METHOD PRIVATE M_Errors : STRING(126)
VAR_INPUT
END_VAR
VAR_INST
END_VAR
CASE _AlarmNum OF	
1	: M_Errors :='1: INTERNAL error';	 	 
2	: M_Errors :='2: No Rtime';	 	 
3	: M_Errors :='3: Allocation locked memory error';	 	 
4	: M_Errors :='4: Insert mailbox error';
5	: M_Errors :='5: Wrong receive HMSG';	 	 
6	: M_Errors :='6: target port NOT found	ADS Server NOT started';	 
7	: M_Errors :='7: target machine NOT found Missing ADS routes';	 
8	: M_Errors :='8: Unknown command ID';	 	 
9	: M_Errors :='9: Bad task ID';	 	 
10	: M_Errors :='10: No IO';	 	 
11	: M_Errors :='11: Unknown ADS command';	 	 
12	: M_Errors :='12: Win 32 error';	 	 
13	: M_Errors :='13: Port NOT connected';	 	 
14	: M_Errors :='14: Invalid ADS length';	 	 
15	: M_Errors :='15: Invalid AMS Net ID';	 	 
16	: M_Errors :='16: Low Installation level';	 	 
17	: M_Errors :='17: No debug available';	 	 
18	: M_Errors :='18: Port disabled';	 	 
19	: M_Errors :='19: Port already connected';	 	 
20	: M_Errors :='20: ADS Sync Win32 error';	 	 
21	: M_Errors :='21: ADS Sync Timeout';	 	 
22	: M_Errors :='22: ADS Sync AMS error';	 	 
23	: M_Errors :='23: ADS Sync no index map';	 	 
24	: M_Errors :='24: Invalid ADS port';	 	 
25	: M_Errors :='25: No memory';	 	 
26	: M_Errors :='26: TCP send error';	 	 
27	: M_Errors :='27: Host unreachable	'; 	 
28	: M_Errors :='28: Invalid AMS fragment';
1101: M_Errors :='';
1792: M_Errors :='1792: error class <device error>';	 	 
1793: M_Errors :='1793: Service is NOT supported BY server';	 	 
1794: M_Errors :='1794: invalid index group';	 	 
1795: M_Errors :='1795: invalid index offset';	 	 
1796: M_Errors :='1796: reading/writing NOT permitted';	 	 
1797: M_Errors :='1797: parameter size NOT correct';	 	 
1798: M_Errors :='1798: invalid parameter value(S)';	 	 
1799: M_Errors :='1799: device is NOT in a ready state';	 	 
1800: M_Errors :='1800: device is busy';	 	 
1801: M_Errors :='1801: invalid context (must be in Windows)';	 	 
1802: M_Errors :='1802: out OF memory';	 	 
1803: M_Errors :='1803: invalid parameter value(S)';	 	 
1804: M_Errors :='1804: NOT found (files, ...)';	 	 
1805: M_Errors :='1805: syntax error in command OR file';	 	 
1806: M_Errors :='1806: objects DO NOT match';	 	 
1807: M_Errors :='1807: object already exists';	 	 
1808: M_Errors :='1808: symbol NOT found';	 	 
1809: M_Errors :='1809: symbol version invalid';	
1810: M_Errors :='1810: server is in invalid state';	 	 
1811: M_Errors :='1811: AdsTransMode NOT supported';	 	 
1812: M_Errors :='1812: notification handle is invalid';	
1813: M_Errors :='1813: notification client NOT registered';	 	 
1814: M_Errors :='1814: no more notification handles';	 	 
1815: M_Errors :='1815: size FOR watch too big';	 	 
1816: M_Errors :='1816: device NOT initialized';	 	 
1817: M_Errors :='1817: device has a timeout';	 	 
1818: M_Errors :='1818: query INTERFACE failed';	 	 
1819: M_Errors :='1819: wrong INTERFACE required';	 	 
1820: M_Errors :='1820: class ID is invalid';	 	 
1821: M_Errors :='1821: object ID is invalid';	 	 
1822: M_Errors :='1822: request is pending';	 	 
1823: M_Errors :='1823: request is aborted';	 	 
1824: M_Errors :='1824: signal warning';	 	 
1825: M_Errors :='1825: invalid ARRAY index';	 	 
1826: M_Errors :='1826: symbol NOT active';	
1827: M_Errors :='1827: access denied';	 	 
1828: M_Errors :='1828: missing license';	 	
1836: M_Errors :='1836: exception occured during system start';	
1856: M_Errors :='1856: Error class <client error>';	 	 
1857: M_Errors :='1857: invalid parameter AT service';	 	 
1858: M_Errors :='1858: polling list is empty';	 	 
1859: M_Errors :='1859: VAR connection already in use';	 	 
1860: M_Errors :='1860: invoke ID in use';	 	 
1861: M_Errors :='1861: timeout elapsed'; 	
1862: M_Errors :='1862: error in win32 subsystem';	 	 
1863: M_Errors :='1863: Invalid client timeout value';	 	 
1864: M_Errors :='1864: ads-port NOT opened';	 	 
1872: M_Errors :='1872: INTERNAL error in ads sync';	 	 
1873: M_Errors :='1873: hash table overflow';	 	 
1874: M_Errors :='1874: key NOT found in hash';	 	 
1875: M_Errors :='1875: no more symbols in cache';	 	 
1876: M_Errors :='1876: invalid response received';	 	 
1877: M_Errors :='1877: sync port is locked';
4096:  M_Errors:=' 4096: INTERNAL error in the REAL-TIME system.';
4097:  M_Errors:=' 4097: Timer value is NOT valid.';
4098:  M_Errors:=' 4098: Task POINTER has the invalid value 0 (zero).';
4099:  M_Errors:=' 4099: Stack POINTER has the invalid value 0 (zero).';
4100:  M_Errors:=' 4100: The request task priority is already assigned.';
4101:  M_Errors:=' 4101: No free TCB (Task Control Block) available. The maximum number OF TCBs is 64.';
4102:  M_Errors:=' 4102: No free semaphores available. The maximum number OF semaphores is 64.';
4103:  M_Errors:=' 4103: No free space available in the queue. The maximum number OF positions in the queue is 64.';
4109:  M_Errors:=' 4109: An external synchronization interrupt is already applied.';
4110:  M_Errors:=' 4110: No external sync interrupt applied.';
4111:  M_Errors:=' 4111: Application OF the external synchronization interrupt has failed.';
4112:  M_Errors:=' 4112: Call OF a service FUNCTION in the wrong context';
4119:  M_Errors:=' 4119: Intel VT-x extension is NOT supported.';
4120:  M_Errors:=' 4120: Intel VT-x extension is NOT enabled in the BIOS.';
4121:  M_Errors:=' 4121: Missing FUNCTION in Intel VT-x extension.';
4122:  M_Errors:=' 4122: Activation OF Intel VT-x fails.';
16384: M_Errors :='16384: INTERNAL error';
16385: M_Errors :='16385: Memory error';
16386: M_Errors :='16386: Nc RETAIN data error (PERSISTENT data)';
16387: M_Errors :='16387: Parameter FOR Monitoring the NC Setpoint Issuing is Invalid';
16388: M_Errors :='16388: External Error';
16400: M_Errors :='16400: Channel identifier NOT allowed';
16401: M_Errors :='16401: Group identifier NOT allowed';
16402: M_Errors :='16402: Axis identifier NOT allowed';
16403: M_Errors :='16403: Encoder identifier NOT allowed';
16404: M_Errors :='16404: Controller identifier NOT allowed';
16405: M_Errors :='16405: Drive identifier NOT allowed';
16406: M_Errors :='16406: Table identifier NOT allowed';
16416: M_Errors :='16416: No PLC-axis INTERFACE during creation OF an axis';
16417: M_Errors :='16417: No axis-PLC INTERFACE during creation OF an axis';
16418: M_Errors :='16418: No encoder-I/O INTERFACE during creation OF an axis';
16419: M_Errors :='16419: No I/O-encoder INTERFACE during creation OF an axis';
16420: M_Errors :='16420: INTERNAL No drive-I/O INTERFACE during creation OF an axis';
16421: M_Errors :='16421: INTERNAL No I/O-drive INTERFACE during creation OF an axis';
16432: M_Errors :='16432: Coupling TYPE NOT allowed';
16434: M_Errors :='16434: Parameter Unknown Channel TYPE';
16448: M_Errors :='16448: Axis is incompatible';
16464: M_Errors :='16464: Channel NOT ready FOR operation';
16465: M_Errors :='16465: Group NOT ready FOR operation';
16466: M_Errors :='16466: Axis NOT ready FOR operation';
16480: M_Errors :='16480: Channel exists';
16481: M_Errors :='16481: Group exists';
16482: M_Errors :='16482: Axis exists';
16483: M_Errors :='16483: Table exists';
16496: M_Errors :='16496: Axis index NOT allowed';
16497: M_Errors :='16497: Axis index NOT allowed';
16641: M_Errors :='16641: Group index NOT allowed';
16642: M_Errors :='16642: Null POINTER';
16643: M_Errors :='16643: No process image';
16644: M_Errors :='16644: M-FUNCTION index NOT allowed';
16645: M_Errors :='16645: No memory';
16646: M_Errors :='16646: NOT ready';
16647: M_Errors :='16647: FUNCTION/command NOT supported';
16648: M_Errors :='16648: Invalid parameter WHILE starting';
16649: M_Errors :='16649: Channel FUNCTION/command NOT executable';
16650: M_Errors :='16650: ItpGoAhead NOT executable';
16656: M_Errors :='16656: Error opening a file';
16657: M_Errors :='16657: Syntax error during loading';
16658: M_Errors :='16658: Syntax error during interpretation';
16659: M_Errors :='16659: Missing subroutine';
16660: M_Errors :='16660: Loading buffer OF interpreter is too small';
16661: M_Errors :='16661: Symbolic - reserved';
16662: M_Errors :='16662: Symbolic - reserved';
16663: M_Errors :='16663: Subroutine incomplete';
16664: M_Errors :='16664: Error WHILE loading the NC PROGRAM';
16665: M_Errors :='16665: Error WHILE loading the NC PROGRAM';
16672: M_Errors :='16672: Divide BY zero';
16673: M_Errors :='16673: Invalid circle parameterization';
16674: M_Errors :='16674: Invalid FPU-Operation';
16688: M_Errors :='16688: Stack overflow: subroutines';
16689: M_Errors :='16689: Stack underflow: subroutines';
16690: M_Errors :='16690: Stack overflow: arithmetic unit';
16691: M_Errors :='16691: Stack underflow: arithmetic unit';
16704: M_Errors :='16704: Register index NOT allowed';
16705: M_Errors :='16705: Unacceptable G-FUNCTION index';
16706: M_Errors :='16706: Unacceptable M-FUNCTION index';
16707: M_Errors :='16707: Unacceptable extended address';
16708: M_Errors :='16708: Unacceptable index TO the INTERNAL H-FUNCTION';
16709: M_Errors :='16709: Machine data value unacceptable';
16720: M_Errors :='16720: Cannot change tool PARAMS here';
16721: M_Errors :='16721: Cannot calculate tool compensation';
16722: M_Errors :='16722: The plane FOR the tool compensation cannot be changed here';
16723: M_Errors :='16723: The D-WORD is missing OR invalid BY turning on the tool compensation';
16724: M_Errors :='16724: The specified tool radius is invalid because the value is <= zero';
16725: M_Errors :='16725: The tool radius cannot be changed here';
16726: M_Errors :='16726: Collision Detection Table is full';
16727: M_Errors :='16727: INTERNAL error WHILE turning on the contour collision detection';
16728: M_Errors :='16728: INTERNAL error within the contour collision detection: update reversed geo failed';
16729: M_Errors :='16729: Unexpected combination OF geometry types BY active contour collision detection';
16730: M_Errors :='16730: Programmed inner circle is smaller than the cutter radius';
16731: M_Errors :='16731: Bottle neck detection recognized contour violation';
16732: M_Errors :='16732: Table FOR corrected entries is full';
16733: M_Errors :='16733: Input table FOR tangential following is full';
16734: M_Errors :='16734: Executing table FOR tangential following is full';
16735: M_Errors :='16735: Geometric entry FOR tangential following cannot be calculated';
16736: M_Errors :='16736: INTERNAL reserved';
16737: M_Errors :='16737: INTERNAL reserved';
16738: M_Errors :='16738: The actual active interpolation rules, zeroshifts, OR rotation cannot be detected';
16752: M_Errors :='16752: Error WHILE loading: Invalid parameter';
16753: M_Errors :='16753: Invalid contour start position';
16754: M_Errors :='16754: Retrace: Invalid INTERNAL entry index';
16755: M_Errors :='16755: Invalid G Code';
16756: M_Errors :='16756: Error WHILE Opening the G Code File';
16896: M_Errors :='16896: Group ID NOT allowed';
16897: M_Errors :='16897: Group TYPE NOT allowed';
16898: M_Errors :='16898: Master axis index NOT allowed';
16899: M_Errors :='16899: Slave axis index NOT ';
16900: M_Errors :='16900: Initializing INTERNAL Error';
16901: M_Errors :='16901: Invalid cycle TIME FOR statement execution task (SAF)';
16903: M_Errors :='16903: Invalid cycle TIME FOR the statement preparation task(SVB)';
16904: M_Errors :='16904: Single step mode NOT allowed';
16905: M_Errors :='16905: Group deactivation NOT allowed';
16906: M_Errors :='16906: Initialization Statement execution state (SAF state) NOT allowed';
16907: M_Errors :='16907: Channel address';
16908: M_Errors :='16908: Axis address (master axis)';
16909: M_Errors :='16909: Master axis address';
16910: M_Errors :='16910: Slave axis address';
16911: M_Errors :='16911: Slave set value generator address';
16912: M_Errors :='16912: Encoder address';
16913: M_Errors :='16913: Controller address';
16914: M_Errors :='16914: Drive address';
16915: M_Errors :='16915: Address Address Master Setpoint Generator';
16916: M_Errors :='16916: Axis INTERFACE NC TO PLC address';
16917: M_Errors :='16917: Slave axis address';
16918: M_Errors :='16918: Table address unknown';
16919: M_Errors :='16919: NcControl address';
16920: M_Errors :='16920: Axis is blocked FOR commands WHILE PERSISTENT NC data are queued';
16921: M_Errors :='16921: The scaling mode MASTER-AUTO-OFFSET is invalid because no REFERENCE table was found';
16922: M_Errors :='16922: The master axis start position does NOT permit synchronization';
16923: M_Errors :='16923: Slave coupling factor (gearing factor) OF 0.0 is NOT allowed';
16924: M_Errors :='16924: Insertion OF master axis into group NOT allowed';
16925: M_Errors :='16925: Deletion OF master axis FROM group NOT allowed'; 
16926: M_Errors :='16926: FUNCTION/feature is NOT supported FROM the setpoint generator';
16927: M_Errors :='16927: Group initialization';
16928: M_Errors :='16928: Group NOT ready / group NOT ready FOR new task';
16929: M_Errors :='16929: Requested set velocity is NOT allowed';
16930: M_Errors :='16930: Requested target position is NOT allowed (master axis)';
16931: M_Errors :='16931: No enable FOR controller AND/OR feed (Master axis)';
16932: M_Errors :='16932: Movement smaller than one encoder increment';
16933: M_Errors :='16933: Drive NOT ready during axis start';
16934: M_Errors :='16934: Invalid parameters OF the emergency stop.';
16935: M_Errors :='16935: The setpoint generator is inactive such that no instructions are accepted';
16936: M_Errors :='16936: Requested traverse distance is NOT allowed';
16937: M_Errors :='16937: Requested target position is NOT allowed (slave axis)';
16938: M_Errors :='16938: No enable FOR controller AND/OR feed (slave axis)';
16939: M_Errors :='16939: The activation position (position threshold) is out OF range OF the actual positioning';
16940: M_Errors :='16940: The start OR activation data OF the external setpoint generation are NOT valid';
16941: M_Errors :='16941: Velocity is NOT CONSTANT';
16942: M_Errors :='16942: Jerk less than OR equal TO 0.0 is NOT allowed';
16943: M_Errors :='16943: Acceleration less than OR equal TO 0.0 is NOT allowed';
16944: M_Errors :='16944: Absolute deceleration value less than OR equal TO 0.0 is NOT allowed';
16945: M_Errors :='16945: Set velocity less than OR equal TO 0.0 is NOT allowed';
16946: M_Errors :='16946: Loss OF precision when trying a positioning';
16947: M_Errors :='16947: Cycle TIME less than OR equal TO 0.0 is NOT allowed';
16948: M_Errors :='16948: PTP data TYPE <intasdouble> range exceeded';
16949: M_Errors :='16949: PTP LHL velocity profile cannot be generated';
16950: M_Errors :='16950: PTP HML velocity profile cannot be generated';
16951: M_Errors :='16951: Start data address is invalid';
16952: M_Errors :='16952: Velocity override (start override) is NOT allowed';
16953: M_Errors :='16953: Start TYPE NOT allowed';
16954: M_Errors :='16954: Velocity overflow (overshoot in the velocity)';
16955: M_Errors :='16955: Start parameter FOR the axis structure is invalid';
16956: M_Errors :='16956: Override generator initialization parameter invalid';
16957: M_Errors :='16957: Slave axis has NOT set value generator';
16958: M_Errors :='16958: Table is empty';
16959: M_Errors :='16959: Table is full';
16960: M_Errors :='16960: No memory available';
16961: M_Errors :='16961: Table already contains an entry';
16962: M_Errors :='16962: Stop is already active';
16963: M_Errors :='16963: Compensation has NOT been carried out over the full compensation section';
16964: M_Errors :='16964: INTERNAL parameters FOR the compensation are invalid';
16965: M_Errors :='16965: Compensation active';
16966: M_Errors :='16966: Compensation NOT active';
16967: M_Errors :='16967: Compensation TYPE invalid';
16968: M_Errors :='16968: Axis address FOR compensation invalid';
16969: M_Errors :='16969: Invalid slave address';
16970: M_Errors :='16970: Coupling velocity invalid';
16971: M_Errors :='16971: Coupling velocities NOT CONSTANT';
16972: M_Errors :='16972: Cycle TIME less than OR equal TO 0.0 is NOT allowed';
16973: M_Errors :='16973: Decoupling task NOT allowed';
16974: M_Errors :='16974: FUNCTION NOT allowed';
16975: M_Errors :='16975: No valid table weighting has been set';
16976: M_Errors :='16976: Axis TYPE, actual position TYPE OR end position TYPE is NOT allowed';
16977: M_Errors :='16977: FUNCTION NOT presently supported';
16978: M_Errors :='16978: State OF state machine invalid';
16979: M_Errors :='16979: REFERENCE cam became free too soon';
16980: M_Errors :='16980: Clearance monitoring between activation OF the hardware latch AND appearance OF the sync pulse';
16981: M_Errors :='16981: No memory available';
16982: M_Errors :='16982: The table slave axis has no active table';
16983: M_Errors :='16983: FUNCTION NOT allowed';
16984: M_Errors :='16984: Stopping compensation NOT allowed';
16985: M_Errors :='16985: Slave table is being used';
16986: M_Errors :='16986: Master OR slave axis is processing a job WHILE coupling is requested';
16987: M_Errors :='16987: Slave (start) parameter is incorrect';
16988: M_Errors :='16988: Slave TYPE is incorrect';
16989: M_Errors :='16989: Axis stop is already active';
16990: M_Errors :='16990: Maximum number OF tables per slave generator reached';
16991: M_Errors :='16991: The scaling mode is invalid';
16992: M_Errors :='16992: Controller enable NOT present';
16993: M_Errors :='16993: Table NOT found';
16994: M_Errors :='16994: Incorrect table TYPE';
16995: M_Errors :='16995: Single step mode';
16996: M_Errors :='16996: Group task unknown (asynchronous table entry)';
16997: M_Errors :='16997: Group FUNCTION unknown (synchronous FUNCTION)';
16998: M_Errors :='16998: Group task FOR slave NOT allowed';
16999: M_Errors :='16999: Group FUNCTION FOR slave NOT allowed';
17000: M_Errors :='17000: FUNCTION NCI Setpoint Generator is Inactive';
17001: M_Errors :='17001: Startposition=Setpoint Position';
17002: M_Errors :='17002: Parameters OF the delay-generator are invalid';
17003: M_Errors :='17003: External parameters OF the superimposed instruction are invalid';
17004: M_Errors :='17004: Invalid override TYPE.';
17005: M_Errors :='17005: Activation position under/overrun';
17006: M_Errors :='17006: Activation impossible: Master is standing';
17007: M_Errors :='17007: Activation mode NOT possible';
17008: M_Errors :='17008: Start parameter FOR the compensation is invalid';
17009: M_Errors :='17009: Start parameter FOR the compensation is invalid';
17010: M_Errors :='17010: Start parameter FOR the compensation is invalid';
17011: M_Errors :='17011: Target position under/overrun';
17012: M_Errors :='17012: Target position will be under/overrun';
17013: M_Errors :='17013: Parameter Group Parameter is Invalid';
17014: M_Errors :='17014: Monitoring Joint Error AT Start OF Setpoint Generation';
17015: M_Errors :='17015: Dynamic parameters NOT permitted';
17017: M_Errors :='17017: The New Target';
17018: M_Errors :='17018: New Velocity FOR Moving OR the FINAL Target Velocity is Invalid';
17019: M_Errors :='17019: The FINAL Velocity OR the New Target Position is Invalid';
17020: M_Errors :='17020: The New Moving Velocity is Invalid';
17021: M_Errors :='17021: INTERNAL Starting Mode is Invalid';
17022: M_Errors :='17022: A requested motion command could NOT be realized';
17023: M_Errors :='17023: The new target position either has been overrun OR will be overrun';
17024: M_Errors :='17024: Group NOT ready / group NOT ready FOR new task';
17025: M_Errors :='17025: The parameters OF the oriented stop (O-Stop) are NOT admitted.';
17026: M_Errors :='17026: The modulo target position OF the modulo-start is invalid';
17027: M_Errors :='17027: The online change activation mode is invalid';
17028: M_Errors :='17028: The parameterized jerk rate is NOT permitted';
17029: M_Errors :='17029: The parameterized acceleration OR deceleration is NOT permitted';
17030: M_Errors :='17030: The parameterized velocity is NOT permitted';
17031: M_Errors :='17031: A activation cannot be executed due TO a pending activation';
17032: M_Errors :='17032: Illegal combination OF different cycle times within an axis group';
17033: M_Errors :='17033: Illegal motion reversal';
17034: M_Errors :='17034: Illegal moment FOR an axis command because there is an old axis command active';
17035: M_Errors :='17035: Error in the stop-calculation routine';
17036: M_Errors :='17036: A command with activation position cannot be performed because the remaining path is too short';
17037: M_Errors :='17037: Illegal decouple TYPE when decoupling a slave axis';
17038: M_Errors :='17038: Illegal target velocity when decoupling a slave axis';
17039: M_Errors :='17039: The command new dynamic parameter cannot be performed since THIS would require a new target velocity';
17040: M_Errors :='17040: A command with activation position cannot be performed because the axis is already in the brake phase';
17041: M_Errors :='17041: Decouple routine OF slave axis does NOT RETURN a valid solution';
17042: M_Errors :='17042: Command NOT be executed because the command buffer is full filled';
17043: M_Errors :='17043: Command is rejected due TO an INTERNAL error in the Look Ahead';
17044: M_Errors :='17044: Command is rejected because the segment target velocity is NOT realized';
17045: M_Errors :='17045: Successive commands have the same FINAL position';
17046: M_Errors :='17046: Logical positioning direction is inconsistent with the direction OF the buffer command';
17047: M_Errors :='17047: Command is rejected because the remaining positioning length is TO small';
17050: M_Errors :='17050: FUNCTION Restart has Failed';
17051: M_Errors :='17051: Collect error FOR invalid start parameters';
17052: M_Errors :='17052: REFERENCE cam is NOT found';
17053: M_Errors :='17053: REFERENCE cam became NOT free';
17054: M_Errors :='17054: IO sync pulse was NOT found (only when using hardware latch)';
17055: M_Errors :='17055: The Used Buffer Mode is Unknown OR NOT Supported in THIS Context';
17056: M_Errors :='17056: Group/axis consequential error';
17057: M_Errors :='17057: Velocity reduction factor FOR C0/C1 transition is NOT allowed';
17058: M_Errors :='17058: Critical angle AT segment transition NOT allowed';
17059: M_Errors :='17059: Radius OF the tolerance sphere';
17060: M_Errors :='17060: Parameter NOT implemented';
17061: M_Errors :='17061: Start TYPE';
17062: M_Errors :='17062: Parameter NOT implemented';
17063: M_Errors :='17063: Blending with given parameters NOT possible';
17064: M_Errors :='17064: Parameter NOT implemented';
17065: M_Errors :='17065: Curve velocity reduction METHOD NOT allowed';
17066: M_Errors :='17066: Minimum velocity NOT allowed';
17067: M_Errors :='17067: Power FUNCTION input NOT allowed';
17068: M_Errors :='17068: Dynamic change parameter NOT allowed';
17069: M_Errors :='17069: Memory allocation error';
17070: M_Errors :='17070: The calculated end position differs FROM the end position in the nc instruction';
17071: M_Errors :='17071: Calculate remaining chord length';
17072: M_Errors :='17072: Set value generator SVB active';
17073: M_Errors :='17073: SVB parameter NOT allowed';
17074: M_Errors :='17074: Velocity reduction factor NOT allowed';
17075: M_Errors :='17075: Helix is a circle';
17076: M_Errors :='17076: Helix is a straight line';
17077: M_Errors :='17077: Guider parameter NOT allowed';
17078: M_Errors :='17078: Invalid segment address';
17079: M_Errors :='17079: Unparameterized generator';
17080: M_Errors :='17080: Unparameterized table';
17082: M_Errors :='17082: The calculation OF the arc length OF the smoothed path failed (INTERNAL error)';
17083: M_Errors :='17083: The radius OF the tolerance ball is too small (smaller than 0.1 mm)';
17084: M_Errors :='17084: INTERNAL Error WHILE calculating DXD-Software-LIMIT switches (INTERNAL error)';
17085: M_Errors :='17085: NC-Block violates software LIMIT switches OF the group';
17086: M_Errors :='17086: INTERNAL error in the evaluation OF a possible software LIMIT switch violation';
17087: M_Errors :='17087: Invalid REFERENCE speed TYPE';
17088: M_Errors :='17088: Interpolating group contains axes OF an incorrect axis TYPE';
17089: M_Errors :='17089: Scalar product cannot be calculated';
17090: M_Errors :='17090: Inverse cosine cannot be calculated';
17091: M_Errors :='17091: Invalid table entry TYPE';
17092: M_Errors :='17092: Invalid DIN66025 information TYPE';
17093: M_Errors :='17093: Invalid dimension';
17094: M_Errors :='17094: Geometrical object is NOT a straight line';
17095: M_Errors :='17095: Geometrical object is NOT a circle';
17096: M_Errors :='17096: Geometrical object is NOT a helix';
17097: M_Errors :='17097: Set velocity less than OR equal TO 0.0 is invalid';
17098: M_Errors :='17098: Address FOR look-ahead invalid';
17099: M_Errors :='17099: Set value generator SAF active';
17100: M_Errors :='17100: CNC set value generation NOT active';
17101: M_Errors :='17101: CNC set value generation in the stop phase';
17102: M_Errors :='17102: Override NOT allowed';
17103: M_Errors :='17103: Invalid table address';
17104: M_Errors :='17104: Invalid table entry TYPE';
17105: M_Errors :='17105: Memory allocation failed';
17106: M_Errors :='17106: Memory allocation failed';
17107: M_Errors :='17107: Invalid parameter';
17108: M_Errors :='17108: Delete Distance TO Go failed';
17109: M_Errors :='17109: The setpoint generator OF the flying saw generates incompatible values (INTERNAL error)';
17110: M_Errors :='17110: Axis will be stopped since otherwise it will overrun its target position';
17111: M_Errors :='17111: INTERNAL error in the transformation FROM slave TO master';
17112: M_Errors :='17112: Wrong direction in the transformation OF slave TO master';
17114: M_Errors :='17114: Parameter OF Motion FUNCTION (MF) table incorrect';
17115: M_Errors :='17115: Parameter OF Motion FUNCTION (MF) table incorrect';
17116: M_Errors :='17116: INTERNAL error BY using Motion FUNCTION (MF)';
17117: M_Errors :='17117: Axis coupling with synchronization generator declined because OF incorrect axis dynamic values';
17118: M_Errors :='17118: Coupling conditions OF synchronization generator incorrect';
17119: M_Errors :='17119: Moving profile OF synchronization generator declines dynamic LIMIT OF slave axis';
17120: M_Errors :='17120: Invalid parameter';
17121: M_Errors :='17121: Invalid parameter';
17122: M_Errors :='17122: External generator is active';
17123: M_Errors :='17123: External generator is NOT active';
17124: M_Errors :='17124: NC-Block with auxiliary axis violates software LIMIT switches OF the group';
17125: M_Errors :='17125: NC-Block TYPE Bezier spline curve contains a cusp (singularity)';
17127: M_Errors :='17127: Value FOR dead TIME compensation NOT allowed';
17128: M_Errors :='17128: GROUPERR_RANGE_NOMOTIONWINDOW';
17129: M_Errors :='17129: GROUPERR_RANGE_NOMOTIONFILTERTIME';
17130: M_Errors :='17130: GROUPERR_RANGE_TIMEUNITFIFO';
17131: M_Errors :='17131: GROUPERR_RANGE_OVERRIDETYPE';
17132: M_Errors :='17132: GROUPERR_RANGE_OVERRIDECHANGETIME';
17133: M_Errors :='17133: GROUPERR_FIFO_INVALIDDIMENSION';
17134: M_Errors :='17134: GROUPERR_ADDR_FIFOTABLE';
17135: M_Errors :='17135: Axis is locked FOR motion commands because a stop command is still active';
17136: M_Errors :='17136: Invalid number OF auxiliary axes';
17137: M_Errors :='17137: Invalid reduction parameter FOR auxiliary axes';
17138: M_Errors :='17138: Invalid dynamic parameter FOR auxiliary axes';
17139: M_Errors :='17139: Invalid coupling parameter FOR auxiliary axes';
17140: M_Errors :='17140: Invalid auxiliary axis entry';
17142: M_Errors :='17142: Invalid parameter';
17144: M_Errors :='17144: Block search - segment NOT found';
17145: M_Errors :='17145: Blocksearch - invalid remaining segment length';
17147: M_Errors :='17147: INTERNAL INTERNAL Error in the Context OF Coupled Axes (Slave Axes)';
17148: M_Errors :='17148: Parameter Parameter FOR the Maximum Number OF Jobs (Entries) TO be Transferred is Invalid';
17151: M_Errors :='17151: Monitoring Customer Specific Error';
17152: M_Errors :='17152: Axis ID NOT allowed';
17153: M_Errors :='17153: Axis TYPE NOT allowed';
17158: M_Errors :='17158: Slow manual velocity NOT allowed';
17159: M_Errors :='17159: Fast manual velocity NOT allowed';
17160: M_Errors :='17160: High speed NOT allowed';
17161: M_Errors :='17161: Acceleration NOT allowed';
17162: M_Errors :='17162: Deceleration NOT allowed';
17163: M_Errors :='17163: Jerk NOT allowed';
17164: M_Errors :='17164: Delay TIME between position AND velocity is NOT allowed';
17165: M_Errors :='17165: Override-TYPE NOT allowed';
17166: M_Errors :='17166: NCI: Velo-Jump-Factor NOT allowed';
17167: M_Errors :='17167: NCI: Radius OF tolerance sphere FOR the auxiliary axes is invalid';
17168: M_Errors :='17168: NCI: Value FOR maximum deviation FOR the auxiliary axes is invalid';
17170: M_Errors :='17170: Referencing velocity in direction OF cam NOT allowed';
17171: M_Errors :='17171: Referencing velocity in sync direction NOT allowed';
17172: M_Errors :='17172: Pulse width in positive direction NOT allowed';
17173: M_Errors :='17173: Pulse width in negative direction NOT allowed';
17174: M_Errors :='17174: Pulse TIME in positive direction NOT allowed';
17175: M_Errors :='17175: Pulse TIME in negative direction NOT allowed';
17176: M_Errors :='17176: Creep distance in positive direction NOT allowed';
17177: M_Errors :='17177: Creep distance in negative direction NOT allowed';
17178: M_Errors :='17178: Braking distance in positive direction NOT allowed';
17179: M_Errors :='17179: Braking distance in negative direction NOT allowed';
17180: M_Errors :='17180: Braking TIME in positive direction NOT allowed';
17181: M_Errors :='17181: Braking TIME in negative direction NOT allowed';
17182: M_Errors :='17182: Switching TIME FROM high TO low speed NOT allowed';
17183: M_Errors :='17183: Creep distance FOR stop NOT allowed';
17184: M_Errors :='17184: Motion monitoring NOT allowed';
17185: M_Errors :='17185: Position window monitoring NOT allowed';
17186: M_Errors :='17186: Target window monitoring NOT allowed';
17187: M_Errors :='17187: Loop NOT allowed';
17188: M_Errors :='17188: Motion monitoring TIME NOT allowed';
17189: M_Errors :='17189: Target window range NOT allowed';
17190: M_Errors :='17190: Position window range NOT allowed';
17191: M_Errors :='17191: Position window monitoring TIME NOT allowed';
17192: M_Errors :='17192: Loop movement NOT allowed';
17193: M_Errors :='17193: Axis cycle TIME NOT allowed';
17194: M_Errors :='17194: Stepper motor operating mode NOT allowed';
17195: M_Errors :='17195: Displacement per stepper motor step NOT allowed';
17196: M_Errors :='17196: Minimum speed FOR stepper motor set value profile NOT allowed';
17197: M_Errors :='17197: Stepper motor stages FOR one speed stage NOT allowed';
17198: M_Errors :='17198: DWORD FOR the interpretation OF the axis units NOT allowed';
17199: M_Errors :='17199: Maximum velocity NOT allowed';
17200: M_Errors :='17200: Motion monitoring window NOT allowed';
17201: M_Errors :='17201: PEH TIME monitoring NOT allowed';
17202: M_Errors :='17202: PEH monitoring TIME NOT allowed';
17203: M_Errors :='17203: Parameter Break Release Delay is Invalid';
17204: M_Errors :='17204: Parameter NC Data Persistence is Invalid';
17205: M_Errors :='17205: Parameter FOR the Error Reaction Mode is Invalid';
17206: M_Errors :='17206: Parameter FOR the Error Reaction Delay is Invalid';
17207: M_Errors :='17207: Parameter “Couple Slave TO Actual Values IF NOT Enabled” is Invalid';
17208: M_Errors :='17208: Parameter Allow Motion Commands TO Slave Axis” is Invalid';
17209: M_Errors :='17209: Parameter Parameter “Allow Motion Commands TO External Setpoint Axis” is Invalid';
17210: M_Errors :='17210: Parameter Parameter “Fading Acceleration” is Invalid';
17211: M_Errors :='17211: Fast Axis Stop Signal TYPE NOT allowed';
17216: M_Errors :='17216: Initialization Parameter Axis initialization';
17217: M_Errors :='17217: Address Parameter Group address';
17218: M_Errors :='17218: Address Parameter Encoder address';
17219: M_Errors :='17219: Address Parameter Controller address';
17220: M_Errors :='17220: Address Parameter Drive address';
17221: M_Errors :='17221: Address Parameter Axis INTERFACE PLC TO NC address';
17222: M_Errors :='17222: Address Parameter Axis INTERFACE NC TO PLC address';
17223: M_Errors :='17223: Address Parameter Size OF axis INTERFACE NC TO PLC is NOT allowed';
17224: M_Errors :='17224: Address Parameter Size OF axis INTERFACE PLC TO NC is NOT allowed';
17238: M_Errors :='17238: Monitoring Parameter Controller enable';
17239: M_Errors :='17239: There is no feed enable FOR negative motion direction';
17240: M_Errors :='17240: Monitoring Parameter Feed enable plus';
17241: M_Errors :='17241: Monitoring Parameter Set velocity NOT allowed';
17242: M_Errors :='17242: Monitoring Parameter Movement smaller than one encoder increment';
17243: M_Errors :='17243: Monitoring Parameter Set acceleration monitoring';
17244: M_Errors :='17244: Monitoring Parameter PEH TIME monitoring';
17245: M_Errors :='17245: Monitoring Parameter Encoder existence monitoring / movement monitoring';
17246: M_Errors :='17246: Monitoring Parameter Looping distance less than breaking distance';
17247: M_Errors :='17247: Monitoring Starting Velocity Invalid';
17248: M_Errors :='17248: Monitoring FINAL Velocity Invalid';
17249: M_Errors :='17249: Monitoring Parameter TIME range exceeded (future)';
17250: M_Errors :='17250: Monitoring Parameter TIME range exceeded (past)';
17251: M_Errors :='17251: Monitoring Parameter Position cannot be determined';
17252: M_Errors :='17252: Monitoring Parameter Position indeterminable (conflicting direction OF travel)';
17264: M_Errors :='17264: Monitoring No Slave Coupling Possible (Velocity Violation)';
17265: M_Errors :='17265: Monitoring No Slave Coupling Possible (Acceleration Violation)';
17266: M_Errors :='17266: Monitoring FINAL Velocity invalid';
17312: M_Errors :='17312: INTERNAL Parameter Axis consequential error';
17408: M_Errors :='17408: Encoder ID NOT allowed';
17409: M_Errors :='17409: Encoder TYPE NOT allowed';
17410: M_Errors :='17410: Encoder mode';
17411: M_Errors :='17411: Encoder counting direction inverted?';
17412: M_Errors :='17412: Referencing status';
17413: M_Errors :='17413: Encoder increments FOR each physical encoder rotation';
17414: M_Errors :='17414: Scaling factor';
17415: M_Errors :='17415: Position offset (zero point offset)';
17416: M_Errors :='17416: Modulo factor';
17417: M_Errors :='17417: Position filter TIME';
17418: M_Errors :='17418: Velocity filter TIME';
17419: M_Errors :='17419: Acceleration filter TIME';
17420: M_Errors :='17420: Cycle TIME NOT allowed';
17422: M_Errors :='17422: Actual position correction / measurement system error correction';
17423: M_Errors :='17423: Filter TIME actual position correction';
17424: M_Errors :='17424: Search direction FOR referencing cam inverted';
17425: M_Errors :='17425: Search direction FOR sync pulse (zero pulse) inverted';
17426: M_Errors :='17426: REFERENCE position';
17427: M_Errors :='17427: Clearance monitoring between activation OF the hardware latch AND appearance OF the sync pulse';
17428: M_Errors :='17428: Minimum clearance between activation OF the hardware latch AND appearance OF the sync pulse';
17429: M_Errors :='17429: External sync pulse';
17430: M_Errors :='17430: Scaling OF the noise rate is NOT allowed';
17431: M_Errors :='17431: Tolerance window FOR modulo-start';
17432: M_Errors :='17432: Encoder REFERENCE mode';
17433: M_Errors :='17433: Encoder evaluation direction';
17434: M_Errors :='17434: Encoder REFERENCE system';
17435: M_Errors :='17435: Encoder position initialization mode';
17436: M_Errors :='17436: Encoder sign interpretation (UNSIGNED- / SIGNED- data TYPE)';
17440: M_Errors :='17440: Software end location monitoring minimum NOT allowed';
17441: M_Errors :='17441: Software end location monitoring maximum NOT allowed';
17442: M_Errors :='17442: Actual value setting is outside the value range';
17443: M_Errors :='17443: Software end location minimum NOT allowed';
17444: M_Errors :='17444: Software end location maximum NOT allowed';
17445: M_Errors :='17445: Filter mask FOR the raw data OF the encoder is invalid';
17446: M_Errors :='17446: REFERENCE mask FOR the raw data OF the encoder is invalid';
17447: M_Errors :='17447: Parameter Parameter Dead TIME Compensation Mode (Encoder) is Invalid';
17448: M_Errors :='17448: Control Bits OF Dead TIME Compensation” (Encoder) is Invalid';
17449: M_Errors :='17449: TIME Related Shift OF Dead TIME Compensation Mode” (Encoder) is Invalid';
17456: M_Errors :='17456: Hardware latch activation (encoder)';
17457: M_Errors :='17457: External hardware latch activation (encoder)';
17458: M_Errors :='17458: External hardware latch activation (encoder)';
17459: M_Errors :='17459: External hardware latch activation (encoder)';
17460: M_Errors :='17460: Encoder FUNCTION NOT supported';
17461: M_Errors :='17461: Encoder FUNCTION is already active';
17472: M_Errors :='17472: Encoder initialization';
17473: M_Errors :='17473: Axis address';
17474: M_Errors :='17474: I/O input structure address';
17475: M_Errors :='17475: I/O output structure address';
17488: M_Errors :='17488: Encoder counter underflow monitoring';
17489: M_Errors :='17489: Encoder counter overflow monitoring';
17504: M_Errors :='17504: Software end location minimum (axis start)';
17505: M_Errors :='17505: Software end location maximum (axis start)';
17506: M_Errors :='17506: Software end location minimum (positioning process)';
17507: M_Errors :='17507: Software end location maximum (positioning process)';
17508: M_Errors :='17508: Encoder hardware error';
17509: M_Errors :='17509: Position initialization error AT system start';
17510: M_Errors :='17510: Invalid IO data FOR more than n subsequent NC cycles';
17511: M_Errors :='17511: Invalid Actual Position (Encoder)';
17512: M_Errors :='17512: Invalid IO Input Data (Error TYPE 1)';
17513: M_Errors :='17513: Invalid IO Input Data (Error TYPE 2)';
17520: M_Errors :='17520: SSI transformation fault OR NOT finished';
17570: M_Errors :='17570: ENCERR_ADDR_CONTROLLER';
17571: M_Errors :='17571: ENCERR_INVALID_CONTROLLERTYPE';
17664: M_Errors :='17664: Controller ID NOT allowed';
17665: M_Errors :='17665: Controller TYPE NOT allowed';
17666: M_Errors :='17666: Controller operating mode NOT allowed';
17667: M_Errors :='17667: Weighting OF the velocity pre-control NOT allowed';
17668: M_Errors :='17668: Following error monitoring (position) NOT allowed';
17669: M_Errors :='17669: Following error (velocity) NOT allowed';
17670: M_Errors :='17670: Following error window (position) NOT allowed';
17671: M_Errors :='17671: Following error filter TIME (position) NOT allowed';
17672: M_Errors :='17672: Following error window (velocity) NOT allowed';
17673: M_Errors :='17673: Following error filter TIME (velocity) NOT allowed';
17674: M_Errors :='17674: Parameter “Controller Output Limitation” Improper';
17680: M_Errors :='17680: Proportional gain Kv OR Kp (controller) NOT allowed';
17681: M_Errors :='17681: Integral-ACTION TIME Tn (controller) NOT allowed';
17682: M_Errors :='17682: Derivative ACTION TIME Tv (controller) NOT allowed';
17683: M_Errors :='17683: Damping TIME Td (controller) NOT allowed';
17684: M_Errors :='17684: Activation OF the automatic offset compensation NOT allowed';
17685: M_Errors :='17685: Additional proportional gain Kv OR Kp (controller) NOT allowed';
17686: M_Errors :='17686: REFERENCE velocity FOR additional proportional gain Kv OR Kp (controller) NOT allowed';
17687: M_Errors :='17687: Proportional gain Pa (proportion) NOT allowed';
17688: M_Errors :='17688: Proportional gain Kv (velocity controller) NOT allowed';
17689: M_Errors :='17689: parameter “Reset TIME Tn (velocity controller) NOT allowed”';
17690: M_Errors :='17690: Parameter Reserved';
17691: M_Errors :='17691: Parameter Reserved';
17692: M_Errors :='17692: Parameter “Velocity Filter TIME” Improper';
17693: M_Errors :='17693: Parameter “Dead zone NOT allowed“';
17695: M_Errors :='17695: Parameter “Proportionality Factor Kcp” Improper';
17696: M_Errors :='17696: parameter ”Rate TIME Tv (velocity controller) NOT allowed”';
17697: M_Errors :='17697: Damping TIME Td (velocity controller) NOT allowed';
17698: M_Errors :='17698: Parameter “Limitation OF the I Part” Improper';
17699: M_Errors :='17699: Parameter “Limitation OF the D Part” Improper';
17700: M_Errors :='17700: Parameter Parameter “Switching Off the I Part During Motion” is Improper';
17701: M_Errors :='17701: Parameter Parameter “Filter TIME FOR P-T2 Filter” Improper';
17702: M_Errors :='17702: Parameter Velocity Observer: “Parameterized Mode” is Improper';
17703: M_Errors :='17703: Parameter Velocity Observer: “Motor Torque CONSTANT Kt OR Kf” is Improper';
17704: M_Errors :='17704: Parameter Velocity Observer: “Motor Moment OF Inertia JM” is Improper';
17705: M_Errors :='17705: Parameter Velocity Observer: “Band Width f0” is Improper';
17706: M_Errors :='17706: Parameter Velocity Observer: “Correction Factor kc” is Improper';
17707: M_Errors :='17707: Parameter Velocity Observer: “TIME CONSTANT T FOR First Order Filter” is Improper';
17708: M_Errors :='17708: Parameter Velocity Observer: “Amplitude Damping d FOR Second Order Filter” is Improper';
17709: M_Errors :='17709: Parameter Velocity Observer: “Frequency fHP OR Frequency fTP FOR Filters OF Second Order” is Improper';
17728: M_Errors :='17728: Controller initialization';
17729: M_Errors :='17729: Axis address';
17730: M_Errors :='17730: Drive address';
17744: M_Errors :='17744: Following error monitoring (position)';
17745: M_Errors :='17745: Following error monitoring (velocity)';
17824: M_Errors :='17824: CONTROLERR_RANGE_AREA_ASIDE';
17825: M_Errors :='17825: CONTROLERR_RANGE_AREA_BSIDE';
17826: M_Errors :='17826: CONTROLERR_RANGE_QNENN';
17827: M_Errors :='17827: CONTROLERR_RANGE_PNENN';
17828: M_Errors :='17828: CONTROLERR_RANGE_AXISIDPRESP0';
17920: M_Errors :='17920: Drive ID NOT allowed';
17921: M_Errors :='17921: Drive TYPE impermissible';
17922: M_Errors :='17922: Drive operating mode impermissible';
17923: M_Errors :='17923: Motor polarity inverted?';
17924: M_Errors :='17924: Drift compensation/speed offset (DAC offset)';
17925: M_Errors :='17925: REFERENCE speed (velocity pre-control)';
17926: M_Errors :='17926: REFERENCE output in percent';
17927: M_Errors :='17927: Quadrant compensation factor';
17928: M_Errors :='17928: Velocity REFERENCE point';
17929: M_Errors :='17929: Output REFERENCE point';
17930: M_Errors :='17930: Minimum OR maximum output limits (output limitation)';
17931: M_Errors :='17931: Parameter "Maximum Value for Output" is Improper';
17932: M_Errors :='17932: Parameter "Internal Drive Control Word" is Improper';
17933: M_Errors :='17933: Parameter "Internal Timer for RESET Behavior of Motion Controller” is Improper';
17934: M_Errors :='17934: Parameter "Master Motion Controller ID" is Improper';
17935: M_Errors :='17935: Drive torque output scaling impermissible';
17936: M_Errors :='17936: Parameter "Drive velocity output scaling is not allowed"';
17937: M_Errors :='17937: Profi Drive DSC proportional gain Kpc (controller) impermissible';
17938: M_Errors :='17938: Table ID is impermissible';
17939: M_Errors :='17939: Table interpolation TYPE is impermissible';
17940: M_Errors :='17940: Output offset in percent is impermissible';
17941: M_Errors :='17941: Profi Drive DSC scaling FOR calculation OF “Xerr” (controller) impermissible';
17942: M_Errors :='17942: Drive acceleration output scaling impermissible';
17943: M_Errors :='17943: Drive position output scaling impermissible';
17944: M_Errors :='17944: Parameter "Dead Time Compensation Mode" (Motion Controller) is Invalid';
17945: M_Errors :='17945: Parameter "Control Bits of Dead Time Compensation" (Motion Controller) is Invalid';
17946: M_Errors :='17946: Parameter "Time Shift of Dead Time Compensation" (Motion Controller) is Invalid';
17947: M_Errors :='17947: Parameter "Output Delay (Velocity)" is Invalid';
17948: M_Errors :='17948: Drive filter TYPE impermissible FOR command variable filter FOR the output position';
17949: M_Errors :='17949: Drive filter TIME impermissible FOR command variable filter FOR the output position';
17950: M_Errors :='17950: Drive filter order impermissible FOR command variable filter FOR the output position';
17952: M_Errors :='17952: BIT mask FOR stepper motor cycle impermissible';
17953: M_Errors :='17953: BIT mask FOR stepper motor holding current impermissible';
17954: M_Errors :='17954: Scaling factor FOR actual torque (actual current) impermissible';
17955: M_Errors :='17955: Filter TIME FOR actual torque is impermissible';
17956: M_Errors :='17956: Filter TIME FOR the temporal derivation OF the actual torque is impermissible';
17957: M_Errors :='17957: Parameter Parameter FOR the “Motion Controller Operation Mode” is Invalid';
17958: M_Errors :='17958: Monitoring Motion Controller Functionality is NOT Supported';
17959: M_Errors :='17959: FUNCTION DRIVEOPERATIONMODEBUSY';
17960: M_Errors :='17960: Monitoring Motion Controller Operation Mode Switching has NOT been configured';
17968: M_Errors :='17968: Overtemperature';
17969: M_Errors :='17969: Undervoltage';
17970: M_Errors :='17970: Wire break in phase A';
17971: M_Errors :='17971: Wire break in phase B';
17972: M_Errors :='17972: Overcurrent in phase A';
17973: M_Errors :='17973: Overcurrent in phase B';
17974: M_Errors :='17974: Torque overload (stall)';
17984: M_Errors :='17984: Drive initialization';
17985: M_Errors :='17985: Axis address';
17986: M_Errors :='17986: Address IO input structure';
17987: M_Errors :='17987: Address IO output structure';
18000: M_Errors :='18000: Drive hardware NOT ready TO operate';
18001: M_Errors :='18001: Monitoring Error in the cyclic communication OF the drive (Life Counter)';
18002: M_Errors :='18002: Changing the table ID when active controller enable is impermissible';
18005: M_Errors :='18005: Invalid IO data FOR more than (n) continuous NC cycles';
18944: M_Errors :='18944: Table ID NOT allowed';
18945: M_Errors :='18945: Table TYPE NOT allowed';
18946: M_Errors :='18946: Number OF lines in the table NOT allowed';
18947: M_Errors :='18947: Number OF columns in the table is NOT allowed';
18948: M_Errors :='18948: Step size (position delta) NOT allowed';
18949: M_Errors :='18949: Period NOT allowed';
18950: M_Errors :='18950: Table is NOT monotonic';
18951: M_Errors :='18951: Table SUB TYPE is NOT allowed';
18952: M_Errors :='18952: Table interpolation TYPE is NOT allowed';
18953: M_Errors :='18953: Incorrect table main TYPE';
18960: M_Errors :='18960: Table initialization';
18961: M_Errors :='18961: NOT enough memory';
18962: M_Errors :='18962: FUNCTION NOT executed, FUNCTION NOT available';
18963: M_Errors :='18963: Line index NOT allowed';
18964: M_Errors :='18964: Column index NOT allowed';
18965: M_Errors :='18965: Number OF lines NOT allowed';
18966: M_Errors :='18966: Number OF columns NOT allowed';
18967: M_Errors :='18967: Error in scaling OR in range entry';
18968: M_Errors :='18968: Multi table slave out OF range';
18969: M_Errors :='18969: Solo table underflow';
18970: M_Errors :='18970: Solo table overflow';
18971: M_Errors :='18971: Incorrect execution mode';
18972: M_Errors :='18972: Impermissible parameter';
18973: M_Errors :='18973: Fifo is empty';
18974: M_Errors :='18974: Fifo is full';
18975: M_Errors :='18975: Point-Index OF Motion FUNCTION invalid';
18976: M_Errors :='18976: No diagonalization OF matrix';
18977: M_Errors :='18977: Number OF spline points TO less';
18978: M_Errors :='18978: Fifo must NOT be overwritten';
18979: M_Errors :='18979: Insufficient number OF Motion FUNCTION points';
19200: M_Errors :='19200: Axis was stopped';
19201: M_Errors :='19201: Axis cannot be started';
19202: M_Errors :='19202: Control mode NOT permitted';
19203: M_Errors :='19203: Axis is NOT moving';
19204: M_Errors :='19204: Invalid Mode';
19205: M_Errors :='19205: Command NOT permitted';
19206: M_Errors :='19206: Parameter incorrect';
19207: M_Errors :='19207: Timeout axis FUNCTION block';
19208: M_Errors :='19208: Axis is in PROTECTED mode';
19209: M_Errors :='19209: Axis is NOT ready';
19210: M_Errors :='19210: Error during referencing';
19211: M_Errors :='19211: Incorrect definition OF the trigger input';
19212: M_Errors :='19212: Position latch was disabled';
19213: M_Errors :='19213: FUNCTION ‘NC status feedback timeout';
19214: M_Errors :='19214: Additional product NOT installed';
19215: M_Errors :='19215: No NC Cycle Counter Update';
19216: M_Errors :='19216: M-FUNCTION query missing';
19217: M_Errors :='19217: Zero offset index is outside the range';
19218: M_Errors :='19218: R-parameter index OR size is invalid';
19219: M_Errors :='19219: Index FOR tool description is invalid';
19220: M_Errors :='19220: Version OF the cyclic channel INTERFACE does NOT match the requested FUNCTION OR the FUNCTION block';
19221: M_Errors :='19221: Channel is NOT ready FOR the requested FUNCTION';
19222: M_Errors :='19222: Requested FUNCTION is NOT activated';
19223: M_Errors :='19223: Axis is already in another group';
19224: M_Errors :='19224: Block search could NOT be executed successfully';
19225: M_Errors :='19225: Invalid block search parameter';
19232: M_Errors :='19232: Cannot ADD all axes';
19248: M_Errors :='19248: POINTER is invalid';
19249: M_Errors :='19249: Memory size invalid';
19250: M_Errors :='19250: Cam table ID is invalid';
19251: M_Errors :='19251: Point ID is invalid';
19252: M_Errors :='19252: Number OF points is invalid';
19253: M_Errors :='19253: MC table TYPE is invalid';
19254: M_Errors :='19254: Number OF rows invalid';
19255: M_Errors :='19255: Number OF columns invalid';
19256: M_Errors :='19256: Step size invalid';
19264: M_Errors :='19264: Terminal TYPE NOT supported';
19265: M_Errors :='19265: Register read/write error';
19266: M_Errors :='19266: Axis is enabled';
19267: M_Errors :='19267: Incorrect size OF the compensation table';
19268: M_Errors :='19268: Parameter The minimum/maximum position in the compensation table does NOT match the position in the table description';
19269: M_Errors :='19269: NOT implemented';
19296: M_Errors :='19296: Motion command did NOT become active';
19297: M_Errors :='19297: Motion command could NOT be monitored BY the PLC';
19298: M_Errors :='19298: Buffered command was terminated with an error';
19299: M_Errors :='19299: Buffered command was completed without feedback';
19300: M_Errors :='19300: BufferMode is NOT supported BY the command';
19301: M_Errors :='19301: Command number is zero';
19302: M_Errors :='19302: FUNCTION block was NOT called cyclically';
19313: M_Errors :='19313: Invalid NCI entry TYPE';
19314: M_Errors :='19314: NCI feed table full';
19315: M_Errors :='19315: FUNCTION INTERNAL error';
19316: M_Errors :='19316: ST_NciTangentialFollowingDesc: tangential axis is NOT an auxiliary axis';
19317: M_Errors :='19317: Parameter ST_NciTangentialFollowingDesc: nPathAxis1 OR nPathAxis2 is NOT a path axis';
19318: M_Errors :='19318: Parameter ST_NciTangentialFollowingDesc: nPathAxis1 AND nPathAxis2 are the same';
19319: M_Errors :='19319: Parameter ST_NciGeoCirclePlane: Circle incorrectly parameterized';
19321: M_Errors :='19321: Monitoring Tangential following: excessively large deviation angle was detected in the current segment';
19322: M_Errors :='19322: FUNCTION NOT implemented';
19323: M_Errors :='19323: Parameter Tangential following: the radius OF the current arc is too small';
19324: M_Errors :='19324: Parameter FB_NciFeedTablePreparation: pEntry is NULL';
19325: M_Errors :='19325: Parameter FB_NciFeedTablePreparation: the specified nEntryType does NOT match the structure TYPE';
19326: M_Errors :='19326: Parameter ST_NciMFuncFast AND ST_NciMFuncHsk: the requested M-FUNCTION is NOT between 0 AND 159';
19327: M_Errors :='19327: Parameter ST_NciDynOvr: the requested value FOR the dynamic override is NOT between 0.01 AND 1';
19328: M_Errors :='19328: Parameter ST_NciVertexSmoothing: invalid parameter';
19329: M_Errors :='19329: Parameter FB_NciFeedTablePrepartion: The requested velocity is NOT in the valid range';
19330: M_Errors :='19330: Parameter ST_Nci*: invalid parameter';
19344: M_Errors :='19344: Parameter Determined drive TYPE is NOT supported';
19345: M_Errors :='19345: Parameter Direction is impermissible';
19346: M_Errors :='19346: SwitchMode is impermissible';
19347: M_Errors :='19347: Mode FOR the parameter handling is impermissible';
19348: M_Errors :='19348: Parameterization OF the torque limits is inconsistent';
19349: M_Errors :='19349: Parameterization OF the position lag LIMIT is impermissible (<=0)';
19350: M_Errors :='19350: Parameterization OF the distance LIMIT is impermissible (<0)';
19351: M_Errors :='19351: An attempt was made TO back up parameters again, although they have already been backed up';
19352: M_Errors :='19352: An attempt was made TO restore parameters, although none have been backed up';
19360: M_Errors :='19360: KinGroup error: the kinematic group is in an error state';
19361: M_Errors :='19361: KinGroup timeout: timeout during call OF a kinematic block';
19376: M_Errors :='19376: The current axis position OR the axis position resulting FROM the new position offset exceeds the valid range OF values';
19377: M_Errors :='19377: The new position offset exceeds the valid range OF values [AX5000: 2^31]';
19378: M_Errors :='19378: The current axis position OR the new position offset falls below the valid range OF values';
19379: M_Errors :='19379: The new position offset falls below the valid range OF values [AX5000: -2^31]';
19380: M_Errors :='19380: The activated feedback AND/OR storage location (AX5000:P-0-0275) differ FROM the parameterization on the FUNCTION block';
19381: M_Errors :='19381: Reinitialisation OF the Nc actual position has failed';
19382: M_Errors :='19382: The command FOR setting OR deleting a position offset has been rejected without sending feedback data';
19383: M_Errors :='19383: The command FOR setting OR deleting a position offset has been rejected with sending feedback data';
19456: M_Errors :='19456: Transformation failed';
19457: M_Errors :='19457: Ambiguous answer';
19458: M_Errors :='19458: Invalid axis position';
19459: M_Errors :='19459: Configuration Invalid dimension';
19460: M_Errors :='19460: NCERR_KINTRAFO_REGISTRATION';
19461: M_Errors :='19461: INTERNAL Newton iteration failed: The Newton iteration does NOT converge';
19462: M_Errors :='19462: INTERNAL Jacobi matrix cannot be inverted';
19463: M_Errors :='19463: Configuration Invalid cascade: THIS kinematic configuration is NOT permitted';
19464: M_Errors :='19464: Programming Singularity: The machine configuration results in singular axis velocities';
19467: M_Errors :='19467: INTERNAL No metainfo: Metainfo POINTER is null';
19475: M_Errors :='19475: Internally NCERR_RBTFRAME_INVALIDWCSTOMCS';
19488: M_Errors :='19488: INTERNAL Transformation failed: Call OF extended kinematic model failed';
19504: M_Errors :='19504: Programming Invalid input frame: Programmed Cartesian position cannot be reached in the ACS configuration';
19536: M_Errors :='19536: Internally Invalid Offset: Access violation within the observer detected';
33024: M_Errors :='33024: INTERNAL error';
33025: M_Errors :='33025: NOT initialized (e.g. no nc axis)';
33026: M_Errors :='33026: Invalid parameter';
33027: M_Errors :='33027: Invalid index offset';
33028: M_Errors :='33028: Invalid parameter size';
33029: M_Errors :='33029: Invalid start parameter (set point generator)';
33030: M_Errors :='33030: NOT supported';
33031: M_Errors :='33031: Nc axis NOT enabled';
33032: M_Errors :='33032: Nc axis in error state';
33033: M_Errors :='33033: IO drive in error state';
33034: M_Errors :='33034: Nc axis AND IO drive in error state';
33035: M_Errors :='33035: Invalid drive operation mode active OR requested (no bode plot mode)';
33036: M_Errors :='33036: Invalid context FOR THIS command (mandatory task OR windows context needed)';
33037: M_Errors :='33037: Missing TCom axis INTERFACE (axis null POINTER)';
33038: M_Errors :='33038: Invalid input cycle counter FROM IO drive (e.g. frozen)';
33039: M_Errors :='33039: Position monitoring: Axis position is outside OF the maximum allowed moving range';
33040: M_Errors :='33040: Driver limitations detected which causes a nonlinear behavior AND invalid results OF the bode plot';
33041: M_Errors :='33041: Life counter monitoring: Lost OF communication TO GUI detected after watchdog timeout is elapsed';
33042: M_Errors :='33042: WC state error (IO data working counter)';
33056: M_Errors :='33056: Invalid configuration FOR Object (e.g. in System Manager)';
33057: M_Errors :='33057: Invalid environment FOR Object (e.g. TcCom-Object Hierarchy OR missing/faulty Objects)';
33058: M_Errors :='33058: Incompatible Driver OR Object';
33072: M_Errors :='33072: Invalid ObjectID OF Communication Target';
33073: M_Errors :='33073: Communication Target expects Call in different Context';
33074: M_Errors :='33074: Invalid State OF Communication Target';
33076: M_Errors :='33076: Communication with Communication Target cannot be established';
33083: M_Errors :='33083: Parameter Transition Mode is invalid';
33084: M_Errors :='33084: Parameter BufferMode is invalid';
33085: M_Errors :='33085: FunctionBlock Only one active Instance OF FUNCTION Block per Group is allowed';
33086: M_Errors :='33086: State Command is NOT allowed in current group state';
33087: M_Errors :='33087: FunctionBlock Slave cannot synchronize';
33088: M_Errors :='33088: Parameter Invalid value FOR one OR more OF the dynamic parameters (Acceleration, Deceleration, Jerk)';
33089: M_Errors :='33089: Parameter IdentInGroup is invalid';
33090: M_Errors :='33090: Parameter The number OF axes in the group is incompatible with the axes convention';
33091: M_Errors :='33091: FUNCTION Block OR respective Command is NOT supported BY Target';
33093: M_Errors :='33093: FunctionBlock Mapping OF Cyclic INTERFACE between Nc AND Plc missing (e.g. AXIS_REF, AXES_GROUP_REF)';
33094: M_Errors :='33094: FunctionBlock Invalid Velocity Value';
33095: M_Errors :='33095: Parameter Invalid Coordinate Dimension';
33096: M_Errors :='33096: FunctionBlock Invalid Input Value';
33097: M_Errors :='33097: Parameter Unsupported Dynamics FOR selected Group Kernel';
33098: M_Errors :='33098: Parameter The programmed position dimension incompatible with the axes convention';
33099: M_Errors :='33099: FunctionBlock Path buffer is invalid. E.g. because provided buffer has invalid address OR is NOT big enough';
33100: M_Errors :='33100: FunctionBlock Path does NOT contain ANY element';
33101: M_Errors :='33101: FunctionBlock Provided Path buffer is too small TO store more Path Elements';
33102: M_Errors :='33102: Parameter Dimension OR AT least one Value OF Transition Parameters is invalid';
33103: M_Errors :='33103: FunctionBlock Invalid OR Incomplete Input ARRAY';
33104: M_Errors :='33104: FunctionBlock Path length is zero';
33105: M_Errors :='33105: State Command is NOT allowed in current axis state';
33106: M_Errors :='33106: State TwinCAT System is shutting down AND cannot complete request';
33107: M_Errors :='33107: Parameter Configured axes convention AND configured axes DO NOT match';
33108: M_Errors :='33108: Initialization Invalid Number OF ACS Axes';
33109: M_Errors :='33109: Initialization Invalid Number OF MCS Data';
33110: M_Errors :='33110: Initialization Invalid Value Set FOR Kinematic Parameters';
33112: M_Errors :='33112: The Given ACS Values Cannot be Reached';
33113: M_Errors :='33113: The Set Target Positions Cannot be Reached';
33120: M_Errors :='33120: Circle Specification in Path is invalid';
33121: M_Errors :='33121: Maximum stream lines reached';
33123: M_Errors :='33123: FunctionBlock Invalid First Segment';
33124: M_Errors :='33124: FunctionBlock Invalid auxiliary point';
33126: M_Errors :='33126: FunctionBlock Invalid parameter FOR GapControlMode';
33127: M_Errors :='33127: External Group got unsupported Axis Event (e.g. State Change)';
33128: M_Errors :='33128: Parameter Unsupported Compensation TYPE';
33130: M_Errors :='33130: Invalid OR no Tracking Transformation';
33133: M_Errors :='33133: Invalid Compensation ObjectId';
33135: M_Errors :='33135: State Coupling would cause a cyclic dependency OF axis (e.g. via MC_GearInPos)';
33136: M_Errors :='33136: FunctionBlock Axis was NOT added TO an axes group, the command is NOT valid';
ELSE
	M_Errors:= 	CONCAT('Undefined Error - ' , TO_STRING( _AlarmNum));
END_CASE
END_METHOD

METHOD PRIVATE M_GetDiagnosis
VAR_INST
	{attribute 'tc_no_symbol'}
	Error				: BOOL;
	ErrorStep			: UINT;
	AdsErrId			: UINT;	
	SercosErrId			: UINT;
	{attribute 'tc_no_symbol'}
	_Step					: UINT;
	{attribute 'tc_no_symbol'} 
	_CmdReadClassXDiag 		: FB_SOEREADCLASSXDIAG;
	{attribute 'tc_no_symbol'} 
	_CmdDiagMessage			: FB_SOEREADDIAGMESSAGE;
	{attribute 'tc_no_symbol'} 
	_CmdDiagNum				: FB_SOEREADDIAGNUMBER;
	{attribute 'tc_no_symbol'} 
	_CmdSoERead				: FB_SOEREAD;
	{attribute 'tc_no_symbol'} 
	_CmdGetSlaveState		: FB_ECGETSLAVESTATE;
	{attribute 'tc_no_symbol'} 
	_CmdReadAmpTemp			: FB_SOEREADAMPLIFIERTEMPERATURE;
	{attribute 'tc_no_symbol'} 
	_CmdReadMotorTemp		: FB_SOEREADMOTORTEMPERATURE;
	{attribute 'tc_no_symbol'} 
	_CmdReadDcBusCurrent	: FB_SOEREADDCBUSCURRENT;
	{attribute 'tc_no_symbol'} 
	_CmdReadDcBusVoltage	: FB_SOEREADDCBUSVOLTAGE;
	{attribute 'tc_no_symbol'} 
	_CmdReadMainVoltage		: FB_SOEAX5000READACTMAINVOLTAGE;	
	{attribute 'tc_no_symbol'} 
	_CmdReadDiagNumList		: FB_SOEREADDIAGNUMBERLIST;
	{attribute 'tc_no_symbol'} 
	_CmdAdsRead			: ADSREAD;
	{attribute 'tc_no_symbol'} 
	readBuffer			: ARRAY[0..9] OF BYTE;
	{attribute 'tc_no_symbol'} 
	Ids					: AMSNETID;
	{attribute 'tc_no_symbol'} 
	_SoEString				: ST_SOE_STRING;

	(* NC-Status *)
	_NCAxisID				: UDINT;

	(* Drive Diag *)
	_DriveType					: STRING(19);
	_MotorType					: STRING(31);
	_DriveStatus				: WORD;
	_Class1Diag					: WORD;
	_stClass1Diag				: ST_AX5000_C1D;
	_stDriveStatus				: ST_AX5000DriveStatus;
	_EcSlaveStateBits			: ST_EcSlaveStateBits;
	_EcSlaveState				: ST_EcSlaveState;
	_PreopToSafeOpError			: BOOL;
	_SafeOpToOpError			: BOOL;
	_CPxInvParamList			: ST_SoE_CPxInvParamList;
	_DiagNumber					: UDINT;
	_DiagNumberList				: ST_SoE_DiagNumList;
	_DiagMessage				: STRING(255);
	
	
	(* Performance Parameters *)	
	_AmpWarningTemp				: UINT;
	_AmpShutdownTemp			: UINT;
	_AmplifierTemperature		: REAL;	
	_MotorWarningTemp			: UINT;
	_MotorShutdownTemp			: UINT;	
	_MotorTemperature			: REAL;
	_DcBusCurrent				: REAL;
	_DcBusVoltage				: REAL;
	_ActMainPeakVoltage			: LREAL;
	_ActMainRMSVoltage			: LREAL;
	
	(* Read variables for conversion from read to actual due to factor difference between read output and drive value *)
	{attribute 'tc_no_symbol'} 
	_AmpWarningTempRead			: UINT;
	{attribute 'tc_no_symbol'} 
	_AmpShutdownTempRead		: UINT;
	{attribute 'tc_no_symbol'} 
	_MotorWarningTempRead		: UINT;
	{attribute 'tc_no_symbol'} 
	_MotorShutdownTempRead		: UINT;	
	{attribute 'tc_no_symbol'} 
	_MotorPeakForceRead 		: UINT;	
END_VAR

VAR CONSTANT
	{attribute 'tc_no_symbol'}
	NCIDXG_AXPARMS			: UDINT := 16#00004000;	(* Axis with ID: Parameter 			*)
	{attribute 'tc_no_symbol'}
	NCIDXO_AXP_HWAMSADDR	: UDINT := 16#00000031;
END_VAR
CASE _Step OF
	0: //Step 0: Idle
		IF Control.SystemTime.SecondPulse THEN
			_Step := 1;
		END_IF
		
	//Step 1-2: Read Class 1 Diagnostics (S-0-011)
	1:	//Step 1: Trigger FB
		_CmdReadClassXDiag(Execute := FALSE, Axis := _Axis);
		_CmdReadClassXDiag(Execute	:= TRUE, DiagClass := 1, Timeout := DEFAULT_ADS_TIMEOUT, Axis := _Axis);
		IF _CmdReadClassXDiag.Busy THEN _Step := 2; END_IF
	
	2:	//Step 2: Write to diagnostic paremeter and check for errors
		_CmdReadClassXDiag(Execute := FALSE, Axis := _Axis);
		IF NOT _CmdReadClassXDiag.Busy THEN 
			IF NOT _CmdReadClassxDiag.Error THEN
				_Class1Diag		:= _CmdReadClassxDiag.ClassXDiag;
				_stClass1Diag 	:= F_ConvWordToSTAX5000C1D(_Class1Diag);
			ELSE 
				Error 		:= TRUE;
				ErrorStep	:= _Step;
				AdsErrId 	:= _CmdReadClassXDiag.AdsErrId; 
				SercosErrId := _CmdReadClassXDiag.SercosErrId;
			END_IF
			_Step	:= 3;
		END_IF
		
	//Step 3-4: Read the diagnose message (S-0-0095) 	
	3:	//Step 3: Trigger FB
		_CmdDiagMessage(Execute := FALSE, Axis := _Axis);
		_CmdDiagMessage(Execute := TRUE, Timeout := DEFAULT_ADS_TIMEOUT,Axis := _Axis);
		IF _CmdDiagMessage.Busy THEN _Step := 4; END_IF		
			
	4:	//Step 4: Write to diagnostic paremeter and check for errors
		_CmdDiagMessage(Execute := FALSE, Axis := _Axis);
		IF NOT _CmdDiagMessage.Busy THEN	
			IF NOT _CmdDiagMessage.Error THEN
				_DiagMessage := LEFT(_CmdDiagMessage.DiagMessage.strData,UINT_TO_INT( _CmdDiagMessage.DiagMessage.iActualSize));
			ELSE 
				Error		:= TRUE;
				ErrorStep	:= _Step;
				AdsErrId 	:= _CmdDiagMessage.AdsErrId; 
				SercosErrId := _CmdDiagMessage.SercosErrId;
			END_IF
			_Step := 5;
		END_IF
		
	//Step 5-6: Read current diagnosis number (S-0-0390)
	5: //Step 5: Trigger FB
		_CmdDiagNum(Execute := FALSE, Axis := _Axis);
		_CmdDiagNum(Execute := TRUE, Timeout := DEFAULT_ADS_TIMEOUT, Axis := _Axis);
		IF _CmdDiagNum.Busy THEN _Step := 6; END_IF
		
	6: //Step 6: Write to diagnostic paremeter and check for errors
		_CmdDiagNum(Execute := FALSE, Axis := _Axis);
		IF NOT _CmdDiagNum.Busy THEN
			IF NOT _CmdDiagNum.Error THEN 
				_DiagNumber := _CmdDiagNum.DiagNumber;
			ELSE 
				Error 		:= TRUE;
				ErrorStep	:= _Step;
				AdsErrId 	:= _CmdDiagNum.AdsErrId;
				SercosErrId := _CmdDiagNum.SercosErrId;
			END_IF
			_Step := 7;
		END_IF

	//Step 7-8: Read drive status word (S-0-0135)
	7:	//Step 7: Trigger read
		_CmdSoERead(Execute :=FALSE, Axis := _Axis);
		_CmdSoERead(Execute	:= TRUE, Idn := 135, Element :=16#44, pDstBuf :=ADR(_DriveStatus), BufLen :=SIZEOF(_DriveStatus), Timeout := DEFAULT_ADS_TIMEOUT, Axis := _Axis,);
		IF _CmdSoERead.Busy THEN _Step := 8; END_IF
		
	8:	//Step 8: Write to diagnostic paremeter and check for errors
		_CmdSoERead(Execute:= FALSE,Axis := _Axis);
		IF NOT _CmdSoERead.Busy THEN			
			IF NOT _CmdSoERead.Error THEN
				_stDriveStatus := F_ConvWordToSTAX5000DriveStatus(_DriveStatus);
			ELSE 
				Error 		:= TRUE;
				ErrorStep	:= _Step;
				AdsErrId 	:= _CmdSoERead.AdsErrId;
				SercosErrId := _CmdSoERead.SercosErrId;
			END_IF
			_Step := 9;
		END_IF
	
	//Step 9-10:	Read drive status ActOpMpdeParNum
	9: //Step 9: Trigger FB
		_CmdSoERead(Execute:= FALSE,Axis := _Axis);	
		_CmdSoERead(Execute	:= TRUE, Idn := _stDriveStatus.iActOpModeParNum, Element :=16#44, pDstBuf :=ADR(_stDriveStatus.eActOpMode), BufLen :=SIZEOF(_stDriveStatus.eActOpMode), Timeout	:= DEFAULT_ADS_TIMEOUT, Axis := _Axis);
		IF _CmdSoERead.Busy THEN _Step := 10; END_IF
			
	10: //Step 10: Check for error
		_CmdSoERead(Execute:= FALSE,Axis := _Axis);
		IF NOT _CmdSoERead.Busy THEN			
			IF NOT _CmdSoERead.Error THEN ; 
			ELSE 
				Error 			:= TRUE;
				ErrorStep		:= _Step;
				AdsErrId 		:= _CmdSoERead.AdsErrId;
				SercosErrId 	:= _CmdSoERead.SercosErrId;
			END_IF
			_Step := 11;
		END_IF

	//Step 11-12: Check for error in state change occured and get invalid parameter list
	11: //Step 11: Trigger FB
		_CmdGetSlaveState(bExecute := FALSE);
		//Get reference from NC
		_CmdAdsRead( PORT := AMSPORT_R0_NC, IDXGRP := NCIDXG_AXPARMS + _Axis.NcToPlc.AxisId, IDXOFFS := NCIDXO_AXP_HWAMSADDR, LEN := SIZEOF(readBuffer), DESTADDR := ADR(readBuffer), READ := TRUE, TMOUT := DEFAULT_ADS_TIMEOUT );
			
		IF NOT _CmdAdsRead.BUSY THEN
			_CmdAdsRead(READ := FALSE);
			_NCAxisID := _Axis.NcToPlc.AxisId;		
			IF NOT _CmdAdsRead.ERR THEN
				MEMCPY(ADR(Ids), ADR(readBuffer), SIZEOF(Ids));														
				MEMCPY(ADR(_DriveRef.nSlaveAddr), ADR(readBuffer[6]), SIZEOF(_DriveRef.nSlaveAddr));  	(* readBuffer[6..7] *)
				MEMCPY(ADR(_DriveRef.nDriveNo), ADR(readBuffer[8]), SIZEOF(_DriveRef.nDriveNo));  		(* readBuffer[8..9] *)		
				_DriveRef.sNetId := F_CreateAmsNetId(Ids);
				_CmdGetSlaveState(sNetID := _DriveRef.sNetId, nSlaveAddr := _DriveRef.nSlaveAddr, bExecute := TRUE, tTimeout := DEFAULT_ADS_TIMEOUT);		
			END_IF
				IF _CmdGetSlaveState.bBusy THEN _Step := 12; END_IF
		END_IF
							
	12: //Step 12: Write to diagnostic paremeter if no errors
		_CmdGetSlaveState(bExecute:= FALSE);
		IF NOT _CmdGetSlaveState.bBusy THEN	
			IF NOT _CmdGetSlaveState.bError THEN 
				_EcSlaveState := _CmdGetSlaveState.state;
				_EcSlaveStateBits := F_ConvSlaveStateToBits(_EcSlaveState);
				ELSE 
					Error 		:= TRUE;
					ErrorStep	:= _Step;
					AdsErrId 	:= UDINT_TO_UINT(_CmdGetSlaveState.nErrId);
			END_IF
			
			// If error in slave read diagnostic word corresponding to appropriate drive state
			IF _EcSlaveStateBits.bError THEN
				IF _EcSlaveStateBits.bPreop THEN
					(* read S-0-0021 - IDN List of Invalid operation data for CP2 (Preop->SaveOp) *)
					MEMSET(ADR(_CPxInvParamList), 0, SIZEOF(_CPxInvParamList));
					_PreopToSafeOpError := TRUE;
					_SafeOpToOpError := FALSE;
					_Step	:= 13;
				ELSIF _EcSlaveStateBits.bSafeOp THEN
					(* read S-0-0022 - IDN List of Invalid operation data for CP3 (SaveOp->Op) *)
					MEMSET(ADR(_CPxInvParamList), 0, SIZEOF(_CPxInvParamList));
					_PreopToSafeOpError := FALSE;
					_SafeOpToOpError := TRUE;
					_Step	:= 15;
				ELSE
					(* Skip S-0-0021 + S-0-0022 *)
					MEMSET(ADR(_CPxInvParamList), 0, SIZEOF(_CPxInvParamList));
					_PreopToSafeOpError := FALSE;
					_SafeOpToOpError := FALSE;
					_Step	:= 17;
				END_IF
			ELSE
				(* Skip S-0-0021 + S-0-0022 *)
				MEMSET(ADR(_CPxInvParamList), 0, SIZEOF(_CPxInvParamList));
				_PreopToSafeOpError := FALSE;
				_SafeOpToOpError := FALSE;
				_Step	:= 19;
			END_IF
		END_IF
		
	// Step 13-14: Read invalid parameter list for IDN S-0-0021 (PreOp->SafeOp) or IDN S-0-0021 (SafeOp->Op) into diagnostic parameter list
	13:	//Step 13: Trigger FB (S-0-0021)
		(* read S22 - IDN List of Invalid operation data for CP3 (SaveOp->Op) *)
		_CmdSoERead(Execute := FALSE, Axis := _Axis);
		_CmdSoERead(Execute := TRUE, Idn := 21, Element := 16#40,pDstBuf := ADR(_CPxInvParamList),BufLen :=SIZEOF(_CPxInvParamList),Timeout	:= DEFAULT_ADS_TIMEOUT, Axis := _Axis);
		IF _CmdSoERead.Busy THEN _Step := 14; END_IF
		
	14:	// Step 14: Check for error
		_CmdSoERead(Execute:= FALSE, Axis := _Axis);
		IF NOT _CmdSoERead.Busy THEN			
			IF NOT _CmdSoERead.Error THEN ;
			ELSE 
				Error 			:= TRUE;
				ErrorStep		:= _Step;
				AdsErrId 		:= _CmdSoERead.AdsErrId;
				SercosErrId		:= _CmdSoERead.SercosErrId;
			END_IF
			_Step	:= 17;
		END_IF
	
	15: //Step 15: Trigger FB (S-0-0022)	
		(* read S22 - IDN List of Invalid operation data for CP3 (SaveOp->Op) *)
		_CmdSoERead( Execute := FALSE, Axis := _Axis);
		_CmdSoERead( Execute := TRUE, Idn := 22, Element := 16#40, pDstBuf := ADR(_CPxInvParamList),BufLen := SIZEOF(_CPxInvParamList), Timeout	:= DEFAULT_ADS_TIMEOUT, Axis := _Axis);
		IF _CmdSoERead.Busy THEN _Step := 16; END_IF
		
	16:	// Step 16: Check for error
		_CmdSoERead(Execute:= FALSE,Axis := _Axis);
		IF NOT _CmdSoERead.Busy THEN		
			IF NOT _CmdSoERead.Error THEN
				;
			ELSE
				Error			:= TRUE;
				ErrorStep		:= _Step;
				AdsErrId		:= _CmdSoERead.AdsErrId;
				SercosErrId		:= _CmdSoERead.SercosErrId;
			END_IF
			_Step	:= 17;
		END_IF
	
	// Step 17-18: Read diagnostic number list
	17:	//Step 17: Trigger FB
		_CmDReadDiagNumList(Execute := FALSE, Axis := _Axis);
		_CmdReadDiagNumList( Execute := TRUE, Timeout := DEFAULT_ADS_TIMEOUT, pDiagNumber := ADR(_DiagNumberList), Size := SIZEOF(_DiagNumberList), Axis := _Axis);
		IF _CmdReadDiagNumList.Busy THEN _Step := 18; END_IF
	
	18: //Step 18: Check for errors and write to diagnostic parameters
		_CmDReadDiagNumList(Execute:= FALSE,Axis := _Axis);
		IF NOT _CmDReadDiagNumList.Busy THEN
			IF  _CmDReadDiagNumList.Error THEN
				Error			:= TRUE;
				ErrorStep		:= _Step;
				AdsErrId		:= _CmDReadDiagNumList.AdsErrId;
				SercosErrId 	:= _CmDReadDiagNumList.SercosErrId;
			END_IF
			_Step := 19;
		END_IF
	
	//Step 19-20: Read configured motor type
	19: //Step 19: Trigger FB
		_CmdSoERead(Execute := FALSE, Axis := _Axis);	
		_CmdSoERead(Execute := TRUE, Idn := P_0_IDNs + 53, Element :=16#44, pDstBuf := ADR(_SoEString), BufLen :=SIZEOF(_SoEString), Timeout := DEFAULT_ADS_TIMEOUT, Axis := _Axis);
		IF _CmdSoERead.Busy THEN _Step := 20; END_IF
		
	20: //Step 20: Check for errors and write to diagnostic parameter
		_CmdSoERead(Execute:= FALSE,Axis := _Axis);
		IF NOT _CmdSoERead.Busy THEN
			
			IF NOT _CmdSoERead.Error THEN
				MEMSET(ADR(_MotorType),0,SIZEOF(_MotorType));
				MEMCPY(ADR(_MotorType),ADR(_SoEString.strData),MIN(SIZEOF(_MotorType),_SoEString.iActualSize));
			ELSE
				Error			:= TRUE;
				ErrorStep		:= _Step;
				AdsErrId		:= _CmdSoERead.AdsErrId;
				SercosErrId		:= _CmdSoERead.SercosErrId;
			END_IF
			_Step	:= 21;
		END_IF
	
	//Step 21-22: Read product code/revision number (P-0-0324)	
	21: //Step 21: Trigger FB
		_CmdSoERead( Execute := FALSE, Axis :=_Axis);	
		_CmdSoERead( Execute := TRUE, Idn := P_0_IDNs + 324, Element :=16#44, pDstBuf :=ADR(_SoEString), BufLen :=SIZEOF(_SoEString), Timeout := DEFAULT_ADS_TIMEOUT, Axis := _Axis);
		IF _CmdSoERead.Busy THEN _Step := 22; END_IF
		
	22: //Step 22: Check for errors and write to diagnositc parameter
		_CmdSoERead(Execute:= FALSE, Axis := _Axis);
		IF NOT _CmdSoERead.Busy THEN	
			IF NOT _CmdSoERead.Error THEN
				MEMSET(ADR(_DriveType),0,SIZEOF(_DriveType));	MEMCPY(ADR(_DriveType),ADR(_SoEString.strData),MIN(SIZEOF(_DriveType),_SoEString.iActualSize));
			ELSE
				Error			:= TRUE;
				ErrorStep		:= _Step;
				AdsErrId		:= _CmdSoERead.AdsErrId;
				SercosErrId		:= _CmdSoERead.SercosErrId;
			END_IF
			_Step := 23;
		END_IF
	
	//Step 23-24: Get amp warning temp (S-0-0200)
	23: //Step 23: Trigger FB
		_CmdSoERead( Execute := FALSE, Axis :=_Axis);	
		_CmdSoERead( Execute := TRUE, Idn := S_0_IDNs + 200, Element :=16#40, pDstBuf :=ADR(_AmpWarningTempRead), BufLen :=SIZEOF(_AmpWarningTempRead), Timeout := DEFAULT_ADS_TIMEOUT, Axis := _Axis);
		IF _CmdSoERead.Busy THEN _Step := 24; END_IF	
	
	24:	//Step 24: Check for errors
		_CmdSoERead(Execute:= FALSE, Axis := _Axis);
		IF NOT _CmdSoERead.Busy THEN	
			IF NOT _CmdSoERead.Error THEN 
				_AmpWarningTemp := _AmpWarningTempRead/10;
			ELSE
				Error			:= TRUE;
				ErrorStep		:= _Step;
				AdsErrId		:= _CmdSoERead.AdsErrId;
				SercosErrId		:= _CmdSoERead.SercosErrId;
			END_IF
			_Step := 25;
		END_IF
	
	//Step 25-26: Get amp shutdown temp (S-0-0203)
	25: //Step 25: Trigger FB
		_CmdSoERead( Execute := FALSE, Axis :=_Axis);	
		_CmdSoERead( Execute := TRUE, Idn := S_0_IDNs + 203, Element :=16#40, pDstBuf :=ADR(_AmpShutdownTempRead), BufLen :=SIZEOF(_AmpShutdownTempRead), Timeout := DEFAULT_ADS_TIMEOUT, Axis := _Axis);
		IF _CmdSoERead.Busy THEN _Step := 26; END_IF		
		
	26:	//Step 26: Check for errors
		_CmdSoERead(Execute:= FALSE, Axis := _Axis);
		IF NOT _CmdSoERead.Busy THEN	
			IF NOT _CmdSoERead.Error THEN 
				_AmpShutdownTemp := _AmpShutdownTempRead/10;
			ELSE
				Error			:= TRUE;
				ErrorStep		:= _Step;
				AdsErrId		:= _CmdSoERead.AdsErrId;
				SercosErrId		:= _CmdSoERead.SercosErrId;
			END_IF
			_Step := 27;
		END_IF
	
	//Step 27-28: Read amplifier temperature (S-0-0384)
	27: //Step 27: Trigger FB
		_CmdReadAmpTemp( Execute := FALSE, Axis := _Axis);
		_CmdReadAmpTemp( Execute := TRUE, Timeout := DEFAULT_ADS_TIMEOUT, Axis := _Axis);
		IF _CmdReadAmpTemp.Busy THEN _Step := 28; END_IF
		
	28:	//Step 28: Check for errors and write to parameter
		_CmdReadAmpTemp( Execute := FALSE, Axis := _Axis);
		IF NOT _CmdReadAmpTemp.Busy THEN
			IF NOT _CmdReadAmpTemp.Error THEN
				_AmplifierTemperature := _CmdReadAmpTemp.AmplifierTemperature;
			ELSE
				Error 		:= TRUE;
				ErrorStep	:= _Step;
				AdsErrId	:= _CmdReadAmpTemp.AdsErrId;
				SercosErrId	:= _CmdReadAmpTemp.SercosErrId;				
			END_IF
			_Step := 29;
		END_IF
		
		
	//Step 29-30: Get motor warning temp (S-0-0201)
	29: //Step 29: Trigger FB
		_CmdSoERead( Execute := FALSE, Axis :=_Axis);	
		_CmdSoERead( Execute := TRUE, Idn := S_0_IDNs + 201, Element :=16#40, pDstBuf :=ADR(_MotorWarningTempRead), BufLen :=SIZEOF(_MotorWarningTempRead), Timeout := DEFAULT_ADS_TIMEOUT, Axis := _Axis);
		IF _CmdSoERead.Busy THEN _Step := 30; END_IF	
	
	30:	//Step 30: Check for errors
		_CmdSoERead(Execute:= FALSE, Axis := _Axis);
		IF NOT _CmdSoERead.Busy THEN	
			IF NOT _CmdSoERead.Error THEN 
				_MotorWarningTemp := _MotorWarningTempRead/10;
			ELSE
				Error			:= TRUE;
				ErrorStep		:= _Step;
				AdsErrId		:= _CmdSoERead.AdsErrId;
				SercosErrId		:= _CmdSoERead.SercosErrId;
			END_IF
			_Step := 31;
		END_IF
	
	//Step 31-32: Get motor shutdown temp (S-0-0204)
	31: //Step 31: Trigger FB
		_CmdSoERead( Execute := FALSE, Axis :=_Axis);	
		_CmdSoERead( Execute := TRUE, Idn := S_0_IDNs + 204, Element :=16#40, pDstBuf :=ADR(_MotorShutdownTempRead), BufLen :=SIZEOF(_MotorShutdownTempRead), Timeout := DEFAULT_ADS_TIMEOUT, Axis := _Axis);
		IF _CmdSoERead.Busy THEN _Step := 32; END_IF		
	32:	//Step 32: Check for errors
		_CmdSoERead(Execute:= FALSE, Axis := _Axis);
		IF NOT _CmdSoERead.Busy THEN	
			IF NOT _CmdSoERead.Error THEN 
				_MotorShutdownTemp := _MotorShutdownTempRead/10;
			ELSE
				Error			:= TRUE;
				ErrorStep		:= _Step;
				AdsErrId		:= _CmdSoERead.AdsErrId;
				SercosErrId		:= _CmdSoERead.SercosErrId;
			END_IF
			_Step := 33;
		END_IF			
		
	//Step 33-34: Read motor temperature (S-0-0383)
	33: //Step 33: Trigger FB
		_CmdReadMotorTemp( Execute := FALSE, Axis := _Axis );
		_CmdReadMotorTemp( Execute := TRUE, Timeout := DEFAULT_ADS_TIMEOUT, Axis := _Axis );
		IF _CmdReadMotorTemp.Busy THEN _Step := 34; END_IF
		
	34: //Step 34: Check for errors and write to diagnostic parameter
		_CmdReadMotorTemp( Execute := FALSE, Axis := _Axis );
		IF NOT _CmdReadMotorTemp.Busy THEN
			IF NOT _CmdReadMotorTemp.Error THEN
				_MotorTemperature 	:= _CmdReadMotorTemp.MotorTemperature;
			ELSE
				Error		 		:= TRUE;
				ErrorStep			:= _Step;
				AdsErrId			:= _CmdReadMotorTemp.AdsErrId;
				SercosErrId			:= _CmdReadMotorTemp.SercosErrId;
			END_IF
			_Step := 35;
		END_IF
		
	//Step 35-36: Read DC bus current (S-0-0381)
	35: //Step 35: Trigger FB
		_CmdReadDcBusCurrent( Execute := FALSE, Axis := _Axis );
		_CmdReadDcBusCurrent( Execute := TRUE, Timeout := DEFAULT_ADS_TIMEOUT, Axis := _Axis );
		IF _CmdReadDcBusCurrent.Busy THEN _Step := 36; END_IF
		
	36: //Step 36: Check for errors and write to diagnostic parameter
		_CmdReadDcBusCurrent( Execute := FALSE, Axis := _Axis );
		IF NOT _CmdReadDcBusCurrent.Busy THEN
			IF NOT _CmdReadDcBusCurrent.Error THEN
				_DcBusCurrent := _CmdReadDcBusCurrent.DcBusCurrent;
			ELSE
				Error 			:= TRUE;
				ErrorStep		:= _Step;
				AdsErrId		:= _CmdReadDcBusCurrent.AdsErrId;
				SercosErrId		:= _CmdReadDcBusCurrent.SercosErrId;
			END_IF
			_Step := 37;
		END_IF
		
	//Step 37-38: Read DC bus voltage (S-0-0380)
	37: //Step 37: Trigger FB
		_CmdReadDcBusVoltage( Execute := FALSE, Axis := _Axis );
		_CmdReadDcBusVoltage( Execute := TRUE, Timeout := DEFAULT_ADS_TIMEOUT, Axis := _Axis );
		IF _CmdReadDcBusVoltage.Busy THEN _Step := 38; END_IF
		
	38: //Step 38: Check for errors and write to diagnostic parameter
		_CmdReadDcBusVoltage( Execute := FALSE, Axis := _Axis );
		IF NOT _CmdReadDcBusVoltage.Busy THEN
			IF NOT _CmdReadDcBusVoltage.Error THEN
				_DcBusVoltage	:= _CmdReadDcBusVoltage.DcBusVoltage;
			ELSE
				Error 			:= TRUE;
				ErrorStep		:= _Step;
				AdsErrId		:= _CmdReadDcBusVoltage.AdsErrId;
				SercosErrId		:= _CmdReadDcBusVoltage.SercosErrId;
			END_IF
			_Step := 39;
		END_IF
		
	//Step 39-40: Read actual main voltage (P-0-0200)
	39: //Step 39: Trigger FB
		_CmdReadMainVoltage( Execute := FALSE, Axis := _Axis );
		_CmdReadMainVoltage( Execute := TRUE, Timeout := DEFAULT_ADS_TIMEOUT, Axis := _Axis );
		IF _CmdReadMainVoltage.Busy THEN _Step := 40; END_IF
		
	40: //Step 40: Check for errors and write to diagnostic parameter
		_CmdReadMainVoltage( Execute := FALSE, Axis := _Axis );
		IF NOT _CmdReadMainVoltage.Busy THEN
			IF NOT _CmdReadMainVoltage.Error THEN
				_ActMainPeakVoltage	:= _CmdReadMainVoltage.ActualMainVoltage;
				_ActMainRMSVoltage	:= _ActMainPeakVoltage/(SQRT(2));	
			ELSE
				Error 				:= TRUE;
				ErrorStep			:= _Step;
				ErrorStep			:= _Step;
				AdsErrId			:= _CmdReadMainVoltage.AdsErrId;
				SercosErrId			:= _CmdReadMainVoltage.SercosErrId;
			END_IF	
			_Step := 41;		
		END_IF
		
	//Step 41-42: Read Safety State (P-0-2002) and set state bool	
	41: //Step 41: Trigger FB
		_CmdSoERead( Execute := FALSE, Axis :=_Axis);	
		_CmdSoERead( Execute := TRUE, Idn := P_0_IDN + 2002, Element :=16#40, pDstBuf :=ADR(_SafetyOptionState), BufLen :=SIZEOF(_SafetyOptionState), Timeout := DEFAULT_ADS_TIMEOUT, Axis := _Axis);
		IF _CmdSoERead.Busy THEN _Step := 42; END_IF
		
	42: //Step 42: Check for errors and write to field parameter
		_CmdSoERead(Execute:= FALSE, Axis := _Axis);
		IF NOT _CmdSoERead.Busy THEN	
			IF NOT _CmdSoERead.Error THEN
				_SafetyStateBool	:= _SafetyOptionState.0;
			ELSE
				Error				:= TRUE;
				ErrorStep			:= _Step;
				AdsErrId			:= _CmdSoERead.AdsErrId;
				SercosErrId			:= _CmdSoERead.SercosErrId;
			END_IF
			_Step := 43;
		END_IF
	
	//Step 43-44: Read torque peak (P-0-0094)	
	43: //Step 43: Trigger FB
		_CmdSoERead( Execute := FALSE, Axis :=_Axis);	
		_CmdSoERead( Execute := TRUE, Idn := P_0_IDN + 92, Element :=16#40, pDstBuf :=ADR(_TorquePeak), BufLen :=SIZEOF(_TorquePeak), Timeout := DEFAULT_ADS_TIMEOUT, Axis := _Axis);
		IF _CmdSoERead.Busy THEN _Step := 44; END_IF
		
	44: //Step 44: Check for errors and write to field parameter
		_CmdSoERead(Execute:= FALSE, Axis := _Axis);
		IF NOT _CmdSoERead.Busy THEN	
			IF NOT _CmdSoERead.Error THEN
				;
			ELSE
				Error			:= TRUE;
				ErrorStep		:= _Step;
				AdsErrId		:= _CmdSoERead.AdsErrId;
				SercosErrId		:= _CmdSoERead.SercosErrId;
			END_IF
			_Step := 45;
		END_IF
		
	//Step 45-46: Read torque feedback percentage (S-0-0084)	
	45: //Step 45: Trigger FB	
		_CmdSoERead( Execute := FALSE, Axis :=_Axis);	
		_CmdSoERead( Execute := TRUE, Idn := S_0_IDNs + 84, Element :=16#40, pDstBuf :=ADR(_TorqueFeedbackPercent), BufLen :=SIZEOF(_TorqueFeedbackPercent), Timeout := DEFAULT_ADS_TIMEOUT, Axis := _Axis);
		IF _CmdSoERead.Busy THEN _Step := 46; END_IF
		
	46: //Step 46: Check for errors and write to field parameter after converting percentage of peak into current Nm
		//Note: In drive manager value read for parameter is real, when read in code however the value returned is an int. i.e. Torque peak - in DM = 6.0, returned from SOE read 6000, Torque % - in DM = 6.7 returned 67. (check date size in IDN description manual for 16 bit or 23 bit size.
		_CmdSoERead(Execute:= FALSE, Axis := _Axis);
		IF NOT _CmdSoERead.Busy THEN	
			IF NOT _CmdSoERead.Error THEN 
				_TorqueFeedback := (INT_TO_REAL(_TorqueFeedbackPercent)/10)*(DINT_TO_LREAL(_TorquePeak)/100000);
			ELSE
				Error			:= TRUE;
				ErrorStep		:= _Step;
				AdsErrId		:= _CmdSoERead.AdsErrId;
				SercosErrId		:= _CmdSoERead.SercosErrId;
			END_IF
			_Step := 47;
		END_IF

	//Step 47-48: Read motor break current (P-0-0064)
	47: //Step 37: Trigger FB
		_CmdSoERead( Execute := FALSE, Axis :=_Axis);	
		_CmdSoERead( Execute := TRUE, Idn := P_0_IDN + 64, Element :=16#40, pDstBuf :=ADR(_ActMotorBreakCurrentRead), BufLen :=SIZEOF(_ActMotorBreakCurrentRead), Timeout := DEFAULT_ADS_TIMEOUT, Axis := _Axis);
		IF _CmdSoERead.Busy THEN _Step := 48; END_IF
		
	48: //Step 48: Check for errors and write to status parameter
		_CmdSoERead(Execute:= FALSE, Axis := _Axis);
		IF NOT _CmdSoERead.Busy THEN	
			IF NOT _CmdSoERead.Error THEN
				_ActMotorBreakCurrent := INT_TO_REAL(_ActMotorBreakCurrentRead)/1000;
			ELSE
				Error			:= TRUE;
				ErrorStep		:= _Step;
				AdsErrId		:= _CmdSoERead.AdsErrId;
				SercosErrId		:= _CmdSoERead.SercosErrId;
			END_IF
			_Step := 49;	
		END_IF
	
	49: //Step 49: Calulate normal torque limit from peak
		_NormalTorqueLimitNm := (UINT_TO_REAL(_NormalTorqueLimit)/100) * (DINT_TO_LREAL(_TorquePeak)/1000);
		_Step := 50;
	
	// Step 50-51: Get motor peak force (P-0-0128)
	50: //Step 50: Trigger FB
		_CmdSoERead( Execute := FALSE, Axis :=_Axis);	
		_CmdSoERead( Execute := TRUE, Idn := P_0_IDN + 128, Element :=16#40, pDstBuf :=ADR(_MotorPeakForceRead), BufLen :=SIZEOF(_MotorPeakForceRead), Timeout := DEFAULT_ADS_TIMEOUT, Axis := _Axis);
		IF _CmdSoERead.Busy THEN _Step := 51; END_IF
		
	51: //Step 48: Check for errors and write to status parameter
		_CmdSoERead(Execute:= FALSE, Axis := _Axis);
		IF NOT _CmdSoERead.Busy THEN	
			IF NOT _CmdSoERead.Error THEN
				_MotorPeakForce := UINT_TO_REAL(_MotorPeakForceRead)/1000;
			ELSE
				Error			:= TRUE;
				ErrorStep		:= _Step;
				AdsErrId		:= _CmdSoERead.AdsErrId;
				SercosErrId		:= _CmdSoERead.SercosErrId;
			END_IF
			_Step		:= 0;	
		END_IF
		
	52: //Display diagnostics function error
		IF Error THEN
			;
		END_IF
END_CASE
END_METHOD

METHOD PRIVATE M_Homing
VAR_INPUT
END_VAR
VAR_INST
             	                			
	_HomingJogPos						: BOOL;	
	{attribute 'tc_no_symbol'}                	                			
	_CMD_Home							: MC_HOME;
	{attribute 'tc_no_symbol'}                	                			
	_CMD_SetPosition					: MC_SETPOSITION;
	{attribute 'tc_no_symbol'}                	                			
	_CMD_SoEAX5000SetPositionOffset		: FB_SoEAX5000SetPositionOffset;
	{attribute 'tc_no_symbol'}   
	_SoEAX5000SetPositionOffsetBusyLatch: BOOL;								//Due to no done bit for function this bit latched on busy then for use in detecting falling edge
	{attribute 'tc_no_symbol'}                	                			
	_CMD_SoEAX5000DeletePositionOffset	: FB_SoEAX5000DeletePositionOffset;
	{attribute 'tc_no_symbol'}                	                				
	_CMD_HomeJOG						: MC_JOG;
	{attribute 'tc_no_symbol'}                	                			
	_R_Trig								: ARRAY[0..6] OF R_TRIG;
END_VAR
// ----------------------------------------
// Homing Outputs
// ----------------------------------------
_HomingEN:=_CMD_Home.Busy OR _CMD_SetPosition.Busy OR _CMD_SoEAX5000SetPositionOffset.Busy;
IF _CMD_Home.Busy OR _CMD_SetPosition.Busy OR _CMD_SoEAX5000SetPositionOffset.Busy THEN _Homed := FALSE; END_IF
IF _CMD_Home.Done OR _CMD_SetPosition.Done OR _R_Trig[1].Q THEN _Homed := TRUE;_SoEAX5000SetPositionOffsetBusyLatch:=FALSE; END_IF

// ----------------------------------------
// Error Handler	
// ----------------------------------------
_r_Trig[0](clk :=
(_CMD_Home.Execute AND _CMD_Home.Error) OR 
(_CMD_SetPosition.Execute AND _CMD_SetPosition.Error) OR
(_CMD_SoEAX5000DeletePositionOffset.Execute AND _CMD_SoEAX5000DeletePositionOffset.Error) OR
(_CMD_SoEAX5000SetPositionOffset.Execute AND _CMD_SoEAX5000SetPositionOffset.Error));


// ----------------------------------------
// Manual Home Selection	
// ----------------------------------------
IF _ManHome.Select AND NOT _ManHome.Interlock THEN
	_ManHome.Select :=TRUE;
ELSE
	_ManHome.Select :=FALSE;
END_IF

IF ((_HomeMode < 3) AND NOT Control.PackMLState.Stopped AND NOT Control.PackMLState.Idle)  THEN
	_ManHome.Messages:= 'Axis Cannot be homed.$LSystem is not in an Stopped or Idle State.';
ELSIF((_HomeMode >= 3) AND NOT Control.PackMLState.Aborted) THEN
	_ManHome.Messages:= 'Axis Cannot be homed as the Machine is not De-energized.$LSystem is not in an Aborted State';
ELSIF _r_Trig[0].Q THEN
	_ManHome.Messages:= 'Axis Homing Error Occurred';
ELSE
	IF (_HomeMode < 3) THEN
		_ManHome.Messages:= 'Axis Ready to be Homed.$LThis will cause motion towards the Switch.';
	ELSE
		_ManHome.Messages:= 'Axis Ready to be Homed.$LThe Axis will remain stationary.';
	END_IF
END_IF


IF _CMD_Home.Done OR _CMD_SetPosition.Done OR _R_Trig[1].Q
	OR ((_HomeMode < 3) AND NOT Control.PackMLState.Stopped AND NOT Control.PackMLState.Idle)
	OR ((_HomeMode >= 3) AND NOT Control.PackMLState.Aborted)
	OR _r_Trig[0].Q THEN
	_ManHome.Interlock :=TRUE; 
ELSE
	_ManHome.Interlock :=FALSE;
END_IF


IF _ManHome.Select  THEN
	_ManHome.Queued :=TRUE;
	_ManHome.Messages:= 'Axis Homing Queued.';
ELSE
	_ManHome.Queued :=FALSE;
END_IF

IF _ManHome.Queued  THEN
	_ManHome.Messages:= 'Axis Homing in Progress.';
	_ManHome.Enabled :=TRUE;
ELSE
	_ManHome.Enabled :=FALSE;
END_IF

// ----------------------------------------
// MC Home	
// ----------------------------------------	
_CMD_Home(
	Axis:= _Axis, 
	Execute:= (_AutoHome OR _ManHome.Enabled) AND _HomeMode <=2,
	HomingMode:= MC_DefaultHoming, 
	BufferMode:= , 
	Options:= , 
	bCalibrationCam:= HomingInput, 
	Done=> , 
	Busy=> , 
	Active=> , 
	CommandAborted=> , 
	Error=> , 
	ErrorID=> );
_R_Trig[3](CLK:=_CMD_Home.Error);IF _R_Trig[3].Q THEN _AlarmNum := _CMD_Home.ErrorID; END_IF	

// ----------------------------------------
// MC Set Position	
// ----------------------------------------			
_CMD_SetPosition(
	Axis:= _Axis, 
	Execute:= (_AutoHome OR _ManHome.Enabled) AND _HomeMode = 3, 
	Position:= _PosMoveHome.Position, 
	Mode:= FALSE, 
	Options:= , 
	Done=> , 
	Busy=> , 
	Error=> , 
	ErrorID=> );	
_R_Trig[4](CLK:=_CMD_SetPosition.Error);IF _R_Trig[4].Q THEN _AlarmNum := _CMD_SetPosition.ErrorID; END_IF	

// ----------------------------------------
// MC Set Position Offset	
// ----------------------------------------		
//* Note to Set P-0-0275 = 2.Use Drive Memory	
_CMD_SoEAX5000SetPositionOffset(
	Execute:= (_AutoHome OR _ManHome.Enabled) AND _HomeMode = 4, 
	Position:= _PosMoveHome.Position, 
	Relative:= FALSE, 
	Feedback:= tc2_mc2_Drive.E_PositionOffsetFeedback.ePositionOffsetFeedback1, 
	Memory:=  tc2_mc2_Drive.E_PositionOffsetMemory.ePositionOffsetMemory_Drive, 
	Busy=> , 
	Error=> , 
	ErrorID=> , 
	Axis:= _Axis);
_R_Trig[5](CLK:=_CMD_SoEAX5000SetPositionOffset.Error);IF _R_Trig[5].Q THEN _AlarmNum := _CMD_SoEAX5000SetPositionOffset.ErrorID; END_IF
IF _CMD_SoEAX5000SetPositionOffset.Busy THEN _SoEAX5000SetPositionOffsetBusyLatch := TRUE; END_IF
_R_Trig[1](CLK:=_SoEAX5000SetPositionOffsetBusyLatch AND NOT _CMD_SoEAX5000SetPositionOffset.Busy);
END_METHOD

METHOD PRIVATE M_Jogging
VAR_INPUT
END_VAR
VAR_INST
	{attribute 'tc_no_symbol'}                	                			
	_accelRate							: LREAL;
	{attribute 'tc_no_symbol'}                	                			
	_decelRate							: LREAL;
	{attribute 'tc_no_symbol'}                	                			
	_jerkTime							: LREAL;
	{attribute 'tc_no_symbol'}                	                			
	_jerkValue							: LREAL;
	{attribute 'tc_no_symbol'}                	                			
	_enableJog							: BOOL;
	{attribute 'tc_no_symbol'}                	                			
	_enableManPos						: BOOL;
	{attribute 'tc_no_symbol'}                	                			
	_manPosAbsActive					: BOOL;
	{attribute 'tc_no_symbol'}                	                			
	_manPosModActive					: BOOL;
	{attribute 'tc_no_symbol'}                	                			
	_manPosRelActive					: BOOL;
	{attribute 'tc_no_symbol'}                	                			
	_CMD_JOG							: MC_JOG;
	{attribute 'tc_no_symbol'}                	                			
	_CMD_MovePosManAbs					: MC_MOVEABSOLUTE;
	{attribute 'tc_no_symbol'}                	                			
	_CMD_MovePosManMod					: MC_MOVEMODULO;
	{attribute 'tc_no_symbol'}                	                			
	_CMD_MovePosManRel					: MC_MOVERELATIVE;
	{attribute 'tc_no_symbol'}                	                			
	_CMD_ManMoveHalt					: MC_HALT;
END_VAR
VAR_INST // added by the converter: edge detectors and wires of the graphical bodies
    _w1, _w2 : BOOL;
    _rt1, _rt2, _rt3, _rt4, _rt5 : R_TRIG;
END_VAR
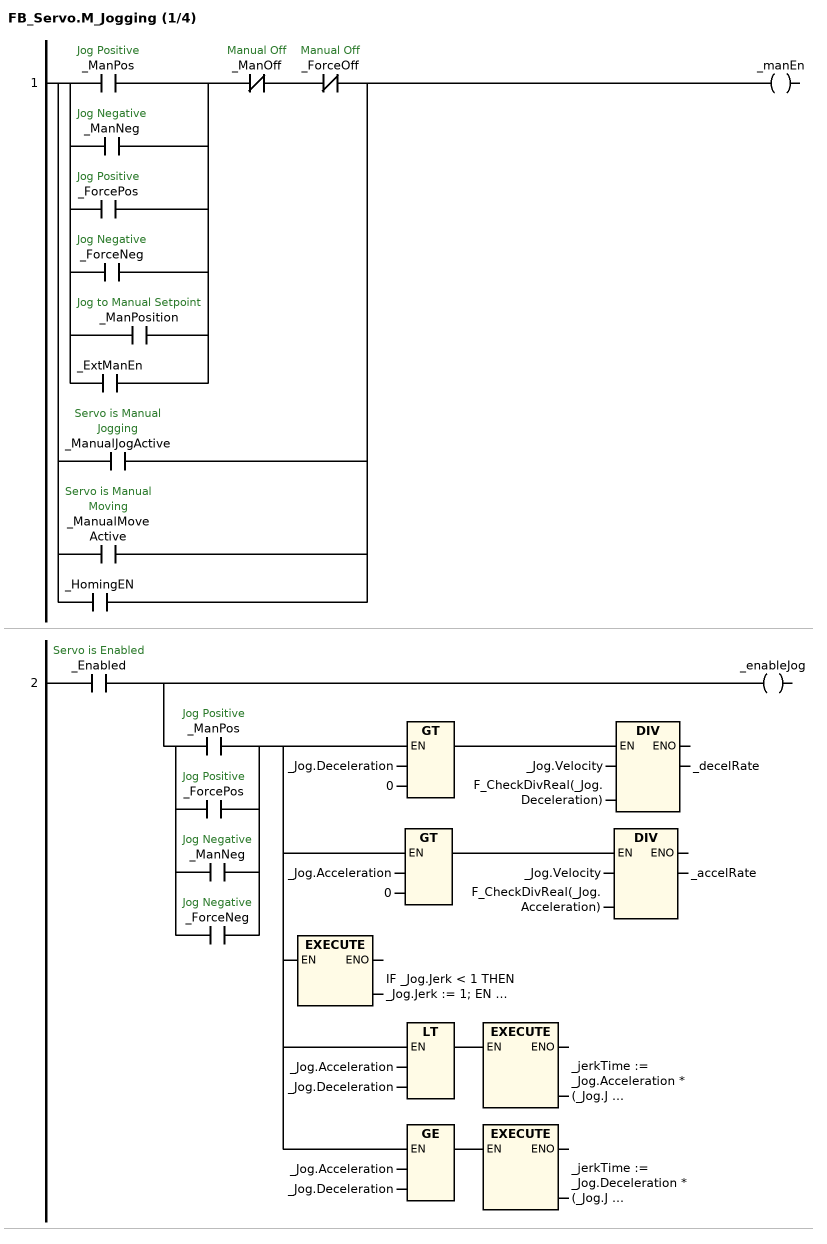
// NETWORK 1
//   _ManPos: Jog Positive
//   _ManNeg: Jog Negative
//   _ForcePos: Jog Positive
//   _ForceNeg: Jog Negative
//   _ManPosition: Jog to Manual Setpoint
//   _ManOff: Manual Off
//   _ForceOff: Manual Off
//   _ManualJogActive: Servo is Manual Jogging
//   _ManualMoveActive: Servo is Manual Moving
_manEn := (_ManPos OR _ManNeg OR _ForcePos OR _ForceNeg OR _ManPosition OR _ExtManEn) AND NOT _ManOff AND NOT _ForceOff OR _ManualJogActive OR _ManualMoveActive OR _HomingEN;

// NETWORK 2
//   _Enabled: Servo is Enabled
//   _ManPos: Jog Positive
//   _ForcePos: Jog Positive
//   _ManNeg: Jog Negative
//   _ForceNeg: Jog Negative
//   _Jog.Velocity: Velocity Value of Move
//   F_CheckDivReal(_Jog.Deceleration): Deceleration Value of Move
//   F_CheckDivReal(_Jog.Acceleration): Accleration Value of Move
//   _Jog.Acceleration: Accleration Value of Move
//   _Jog.Deceleration: Deceleration Value of Move
_enableJog := _Enabled;
_w1 := _Enabled AND (_ManPos OR _ForcePos OR _ManNeg OR _ForceNeg);
IF _w1 AND _Jog.Deceleration > 0 THEN _decelRate := _Jog.Velocity / (F_CheckDivReal(_Jog.Deceleration)); END_IF
IF _w1 AND _Jog.Acceleration > 0 THEN _accelRate := _Jog.Velocity / (F_CheckDivReal(_Jog.Acceleration)); END_IF
IF _w1 THEN
    IF _Jog.Jerk < 1 THEN _Jog.Jerk := 1; END_IF
    IF _Jog.Jerk > 100 THEN _Jog.Jerk := 100; END_IF
END_IF
IF _w1 AND _Jog.Acceleration < _Jog.Deceleration THEN
    _jerkTime := _Jog.Acceleration * (_Jog.Jerk / 100);
    IF _jerkTime > 0 THEN
    	_jerkValue := _accelRate / F_CheckDivReal(LREAL_TO_REAL(_jerkTime));
    END_IF
END_IF
IF _w1 AND _Jog.Acceleration >= _Jog.Deceleration THEN
    _jerkTime := _Jog.Deceleration * (_Jog.Jerk / 100);
    IF _jerkTime > 0 THEN
    	_jerkValue := _decelRate / F_CheckDivReal(LREAL_TO_REAL(_jerkTime));
    END_IF
END_IF

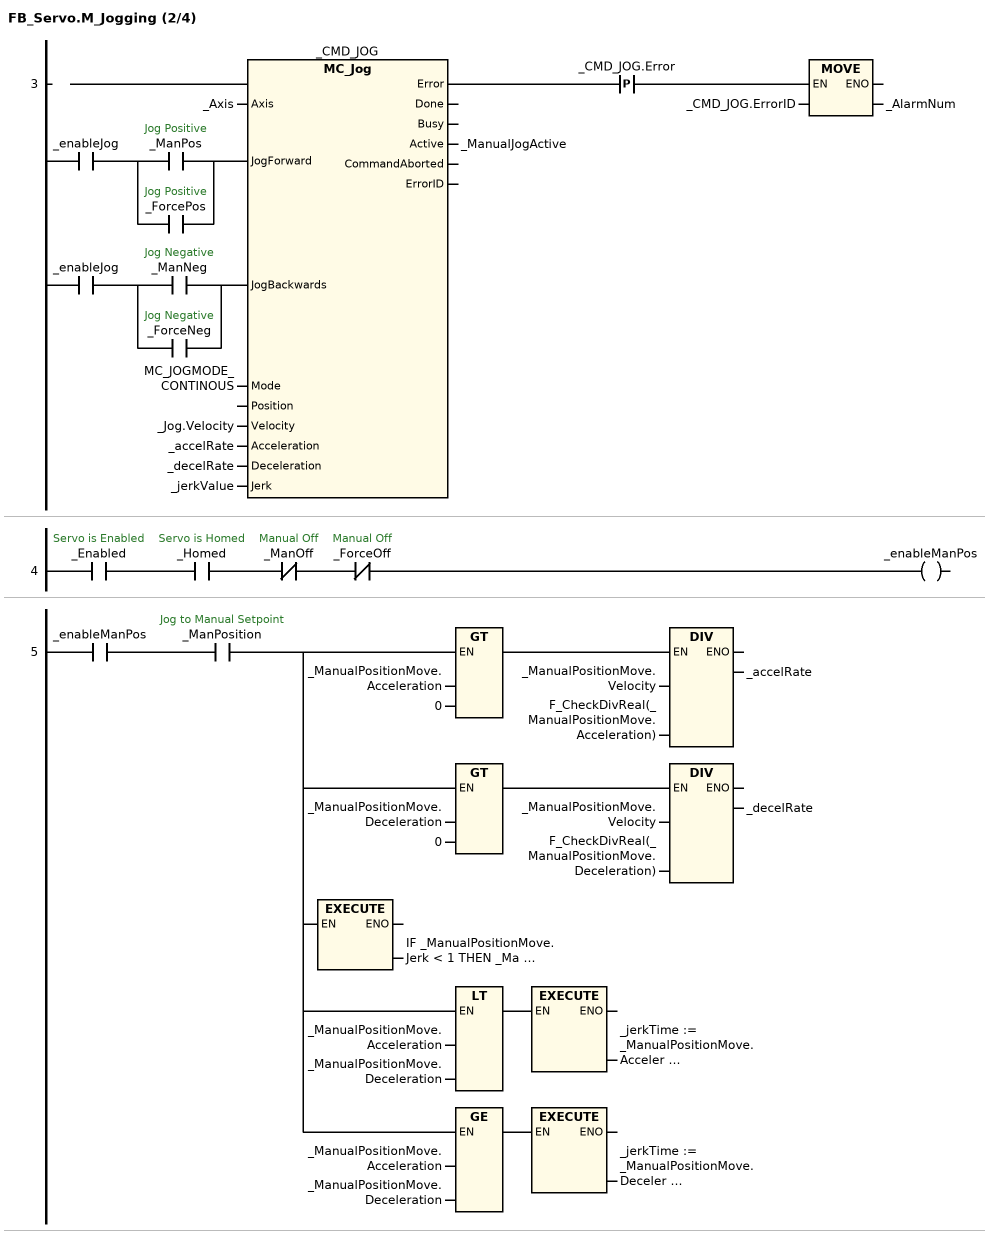
// NETWORK 3
//   _ManPos: Jog Positive
//   _ForcePos: Jog Positive
//   _ManNeg: Jog Negative
//   _ForceNeg: Jog Negative
//   MC_JOGMODE_CONTINOUS: axis moves as long as the jog button is pressed using parameterized dynamics
//   _Jog.Velocity: Velocity Value of Move
//   _ManualJogActive: Servo is Manual Jogging
_CMD_JOG(
    Axis := _Axis,
    JogForward := _enableJog AND (_ManPos OR _ForcePos),
    JogBackwards := _enableJog AND (_ManNeg OR _ForceNeg),
    Mode := MC_JOGMODE_CONTINOUS,
    Velocity := _Jog.Velocity,
    Acceleration := _accelRate,
    Deceleration := _decelRate,
    Jerk := _jerkValue,
    Active => _ManualJogActive); // MC_Jog
_rt1(CLK := _CMD_JOG.Error);
IF _CMD_JOG.Error AND _rt1.Q THEN _AlarmNum := _CMD_JOG.ErrorID; END_IF

// NETWORK 4
//   _Enabled: Servo is Enabled
//   _Homed: Servo is Homed
//   _ManOff: Manual Off
//   _ForceOff: Manual Off
_enableManPos := _Enabled AND _Homed AND NOT _ManOff AND NOT _ForceOff;

// NETWORK 5
//   _ManPosition: Jog to Manual Setpoint
//   _ManualPositionMove.Velocity: Velocity Value of Move
//   F_CheckDivReal(_ManualPositionMove.Acceleration): Accleration Value of Move
//   F_CheckDivReal(_ManualPositionMove.Deceleration): Deceleration Value of Move
//   _ManualPositionMove.Acceleration: Accleration Value of Move
//   _ManualPositionMove.Deceleration: Deceleration Value of Move
_w2 := _enableManPos AND _ManPosition;
IF _w2 AND _ManualPositionMove.Acceleration > 0 THEN
    _accelRate := _ManualPositionMove.Velocity / (F_CheckDivReal(_ManualPositionMove.Acceleration));
END_IF
IF _w2 AND _ManualPositionMove.Deceleration > 0 THEN
    _decelRate := _ManualPositionMove.Velocity / (F_CheckDivReal(_ManualPositionMove.Deceleration));
END_IF
IF _w2 THEN
    IF _ManualPositionMove.Jerk < 1 THEN _ManualPositionMove.Jerk := 1; END_IF
    IF _ManualPositionMove.Jerk > 100 THEN _ManualPositionMove.Jerk := 100; END_IF
END_IF
IF _w2 AND _ManualPositionMove.Acceleration < _ManualPositionMove.Deceleration THEN
    _jerkTime := _ManualPositionMove.Acceleration * (_ManualPositionMove.Jerk / 100);
    IF _jerkTime > 0 THEN
    	_jerkValue := _accelRate / F_CheckDivReal(LREAL_TO_REAL(_jerkTime));
    END_IF
END_IF
IF _w2 AND _ManualPositionMove.Acceleration >= _ManualPositionMove.Deceleration THEN
    _jerkTime := _ManualPositionMove.Deceleration * (_ManualPositionMove.Jerk / 100);
    IF _jerkTime > 0 THEN
    	_jerkValue := _decelRate / F_CheckDivReal(LREAL_TO_REAL(_jerkTime));
    END_IF
END_IF

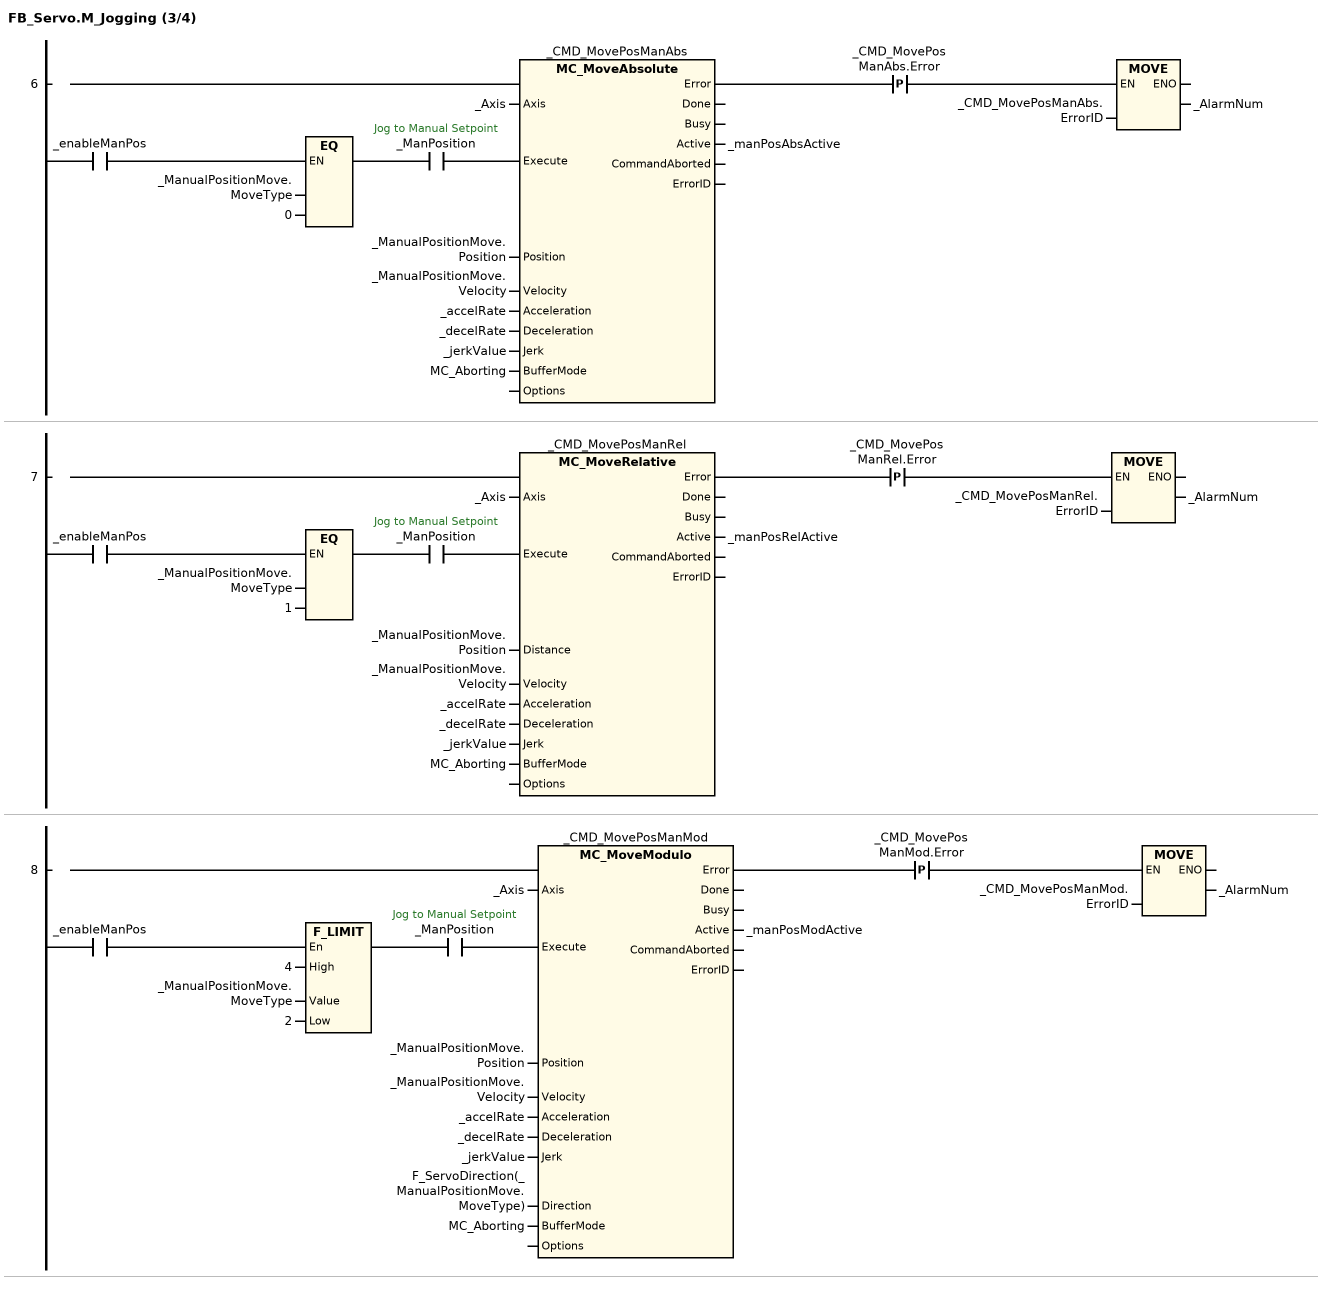
// NETWORK 6
//   _ManualPositionMove.MoveType: Move Type Configuration of Positional Move
//   _ManPosition: Jog to Manual Setpoint
//   _ManualPositionMove.Position: Position Value to Move to
//   _ManualPositionMove.Velocity: Velocity Value of Move
_CMD_MovePosManAbs(
    Axis := _Axis,
    Execute := (_enableManPos AND _ManualPositionMove.MoveType = 0) AND _ManPosition,
    Position := _ManualPositionMove.Position,
    Velocity := _ManualPositionMove.Velocity,
    Acceleration := _accelRate,
    Deceleration := _decelRate,
    Jerk := _jerkValue,
    BufferMode := MC_Aborting,
    Active => _manPosAbsActive); // MC_MoveAbsolute
_rt2(CLK := _CMD_MovePosManAbs.Error);
IF _CMD_MovePosManAbs.Error AND _rt2.Q THEN _AlarmNum := _CMD_MovePosManAbs.ErrorID; END_IF

// NETWORK 7
//   _ManualPositionMove.MoveType: Move Type Configuration of Positional Move
//   _ManPosition: Jog to Manual Setpoint
//   _ManualPositionMove.Position: Position Value to Move to
//   _ManualPositionMove.Velocity: Velocity Value of Move
_CMD_MovePosManRel(
    Axis := _Axis,
    Execute := (_enableManPos AND _ManualPositionMove.MoveType = 1) AND _ManPosition,
    Distance := _ManualPositionMove.Position,
    Velocity := _ManualPositionMove.Velocity,
    Acceleration := _accelRate,
    Deceleration := _decelRate,
    Jerk := _jerkValue,
    BufferMode := MC_Aborting,
    Active => _manPosRelActive); // MC_MoveRelative
_rt3(CLK := _CMD_MovePosManRel.Error);
IF _CMD_MovePosManRel.Error AND _rt3.Q THEN _AlarmNum := _CMD_MovePosManRel.ErrorID; END_IF

// NETWORK 8
//   _ManualPositionMove.MoveType: Move Type Configuration of Positional Move
//   _ManPosition: Jog to Manual Setpoint
//   _ManualPositionMove.Position: Position Value to Move to
//   _ManualPositionMove.Velocity: Velocity Value of Move
_CMD_MovePosManMod(
    Axis := _Axis,
    Execute := F_LIMIT(En := _enableManPos, High := 4, Value := _ManualPositionMove.MoveType, Low := 2) AND _ManPosition,
    Position := _ManualPositionMove.Position,
    Velocity := _ManualPositionMove.Velocity,
    Acceleration := _accelRate,
    Deceleration := _decelRate,
    Jerk := _jerkValue,
    Direction := F_ServoDirection(_ManualPositionMove.MoveType),
    BufferMode := MC_Aborting,
    Active => _manPosModActive); // MC_MoveModulo
_rt4(CLK := _CMD_MovePosManMod.Error);
IF _CMD_MovePosManMod.Error AND _rt4.Q THEN _AlarmNum := _CMD_MovePosManMod.ErrorID; END_IF

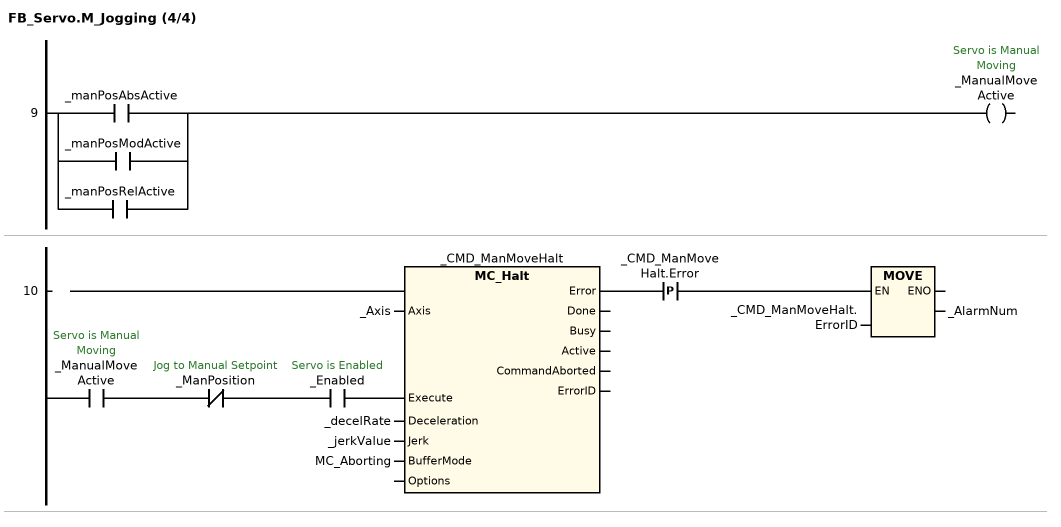
// NETWORK 9
//   _ManualMoveActive: Servo is Manual Moving
_ManualMoveActive := _manPosAbsActive OR _manPosModActive OR _manPosRelActive;

// NETWORK 10
//   _ManualMoveActive: Servo is Manual Moving
//   _ManPosition: Jog to Manual Setpoint
//   _Enabled: Servo is Enabled
_CMD_ManMoveHalt(
    Axis := _Axis,
    Execute := _ManualMoveActive AND NOT _ManPosition AND _Enabled,
    Deceleration := _decelRate,
    Jerk := _jerkValue,
    BufferMode := MC_Aborting); // MC_Halt
_rt5(CLK := _CMD_ManMoveHalt.Error);
IF _CMD_ManMoveHalt.Error AND _rt5.Q THEN _AlarmNum := _CMD_ManMoveHalt.ErrorID; END_IF
END_METHOD

